C03631=1012.728,1.507,383.376,-29.710,62.357,-30.586
C03632=1012.729,1.110,383.407,-29.703,62.283,-30.592
C03633=1012.732,0.714,383.438,-29.696,62.210,-30.597
C03634=1012.733,0.320,383.469,-29.689,62.138,-30.603
C03635=1012.735,-0.076,383.499,-29.682,62.066,-30.609
C03636=1012.736,-0.474,383.530,-29.675,61.994,-30.616
C03637=1012.738,-0.874,383.560,-29.669,61.922,-30.622
C03638=1012.740,-1.277,383.591,-29.662,61.851,-30.627
C03639=1012.742,-1.681,383.623,-29.655,61.779,-30.634
C03640=1012.744,-2.088,383.654,-29.648,61.709,-30.640
C03641=1012.745,-2.496,383.686,-29.642,61.639,-30.646
C03642=1012.746,-2.906,383.717,-29.635,61.568,-30.653
C03643=1012.748,-3.317,383.749,-29.629,61.499,-30.660
C03644=1012.750,-3.719,383.781,-29.623,61.431,-30.667
C03645=1012.751,-4.104,383.810,-29.618,61.367,-30.674
C03646=1012.753,-4.484,383.839,-29.612,61.304,-30.679
C03647=1012.754,-4.874,383.869,-29.606,61.241,-30.686
C03648=1012.756,-5.289,383.902,-29.600,61.175,-30.693
C03649=1012.757,-5.503,383.919,-29.597,61.140,-30.697
C03650=1012.757,-5.720,383.935,-29.594,61.106,-30.699
C03651=1012.758,-5.936,383.952,-29.591,61.072,-30.704
C03652=1012.760,-6.154,383.969,-29.588,61.037,-30.708
C03653=1012.760,-6.370,383.986,-29.585,61.003,-30.710
C03654=1012.761,-6.586,384.002,-29.582,60.969,-30.715
C03655=1012.761,-6.803,384.019,-29.579,60.936,-30.719
C03656=1012.763,-7.019,384.036,-29.576,60.903,-30.722
C03657=1012.763,-7.233,384.052,-29.573,60.870,-30.726
C03658=1012.764,-7.448,384.069,-29.571,60.838,-30.730
C03659=1012.765,-7.661,384.085,-29.568,60.805,-30.734
C03660=1012.766,-7.874,384.102,-29.565,60.773,-30.736
C03661=1012.766,-8.086,384.118,-29.563,60.742,-30.742
C03662=1012.767,-8.297,384.135,-29.560,60.710,-30.745
C03663=1012.768,-8.509,384.150,-29.557,60.679,-30.748
C03664=1012.769,-8.721,384.167,-29.555,60.648,-30.752
C03665=1012.769,-8.932,384.183,-29.552,60.618,-30.756
C03666=1012.770,-9.143,384.200,-29.550,60.587,-30.759
C03667=1012.772,-9.564,384.233,-29.545,60.526,-30.767
C03668=1012.773,-9.986,384.265,-29.540,60.466,-30.775
C03669=1012.775,-10.407,384.298,-29.534,60.407,-30.781
C03670=1012.776,-10.827,384.331,-29.530,60.348,-30.789
C03671=1012.778,-11.244,384.363,-29.525,60.292,-30.796
C03672=1012.779,-11.662,384.395,-29.521,60.235,-30.804
C03673=1012.780,-12.078,384.427,-29.516,60.179,-30.811
C03674=1012.782,-12.491,384.459,-29.512,60.125,-30.818
C03675=1012.783,-12.903,384.491,-29.507,60.071,-30.825
C03676=1012.784,-13.307,384.523,-29.503,60.020,-30.833
C03677=1012.786,-13.699,384.553,-29.499,59.970,-30.839
C03678=1012.787,-14.081,384.582,-29.495,59.922,-30.846
C03679=1012.788,-14.456,384.611,-29.492,59.877,-30.853
C03680=1012.789,-14.832,384.640,-29.488,59.831,-30.859
C03681=1012.790,-15.211,384.670,-29.485,59.785,-30.866
C03682=1012.791,-15.599,384.700,-29.481,59.740,-30.873
C03683=1012.792,-15.994,384.730,-29.478,59.694,-30.880
C03684=1012.793,-16.390,384.761,-29.474,59.648,-30.887
C03685=1012.795,-16.786,384.791,-29.471,59.603,-30.894
C03686=1012.796,-17.184,384.822,-29.468,59.560,-30.901
C03687=1012.797,-17.573,384.852,-29.464,59.517,-30.907
C03688=1012.797,-17.970,384.884,-29.461,59.474,-30.914
C03689=1012.798,-18.197,384.901,-29.459,59.449,-30.917
C03690=1012.799,-18.450,384.920,-29.457,59.423,-30.922
C03691=1012.800,-18.721,384.942,-29.455,59.394,-30.926
C03692=1012.800,-19.000,384.964,-29.453,59.366,-30.931
C03693=1012.801,-19.275,384.984,-29.451,59.338,-30.936
C03694=1012.802,-19.532,385.004,-29.449,59.312,-30.941
C03695=1012.803,-19.762,385.022,-29.448,59.289,-30.944
C03696=1012.802,-19.967,385.038,-29.446,59.269,-30.948
C03697=1012.804,-20.318,385.065,-29.444,59.235,-30.954
C03698=1012.804,-20.714,385.096,-29.441,59.196,-30.961
C03699=1012.806,-21.107,385.127,-29.439,59.160,-30.967
C03700=1012.806,-21.501,385.157,-29.436,59.123,-30.974
C03701=1012.808,-21.894,385.187,-29.433,59.087,-30.980
C03702=1012.809,-22.287,385.218,-29.431,59.052,-30.987
C03703=1012.809,-22.680,385.248,-29.429,59.018,-30.992
C03704=1012.810,-23.074,385.279,-29.426,58.985,-30.999
C03705=1012.811,-23.467,385.308,-29.424,58.951,-31.005
C03706=1012.811,-23.860,385.339,-29.422,58.919,-31.013
C03707=1012.812,-24.253,385.370,-29.420,58.887,-31.019
C03708=1012.813,-24.646,385.401,-29.418,58.858,-31.024
C03709=1012.815,-25.040,385.430,-29.416,58.827,-31.031
C03710=1012.815,-25.433,385.461,-29.415,58.798,-31.037
C03711=1012.816,-25.827,385.492,-29.413,58.768,-31.043
C03712=1012.816,-26.219,385.522,-29.411,58.741,-31.049
C03713=1012.817,-26.613,385.552,-29.410,58.714,-31.055
C03714=1012.818,-27.007,385.583,-29.408,58.687,-31.062
C03715=1012.819,-27.399,385.613,-29.407,58.661,-31.067
C03716=1012.819,-27.793,385.644,-29.405,58.636,-31.073
C03717=1012.820,-28.186,385.674,-29.404,58.611,-31.079
C03718=1012.820,-28.580,385.705,-29.403,58.588,-31.084
C03719=1012.821,-28.973,385.735,-29.401,58.565,-31.090
C03720=1012.822,-29.366,385.766,-29.400,58.541,-31.096
C03721=1012.823,-29.760,385.796,-29.399,58.520,-31.101
C03722=1012.823,-30.153,385.826,-29.398,58.499,-31.106
C03723=1012.823,-30.547,385.857,-29.397,58.479,-31.113
C03724=1012.824,-30.940,385.888,-29.396,58.459,-31.118
C03725=1012.825,-31.333,385.918,-29.396,58.440,-31.124
C03726=1012.825,-31.727,385.948,-29.394,58.422,-31.128
C03727=1012.826,-32.120,385.979,-29.394,58.404,-31.135
C03728=1012.826,-32.514,386.010,-29.393,58.388,-31.138
C03729=1012.826,-32.907,386.040,-29.393,58.372,-31.144
C03730=1012.827,-33.301,386.070,-29.393,58.357,-31.149
C03731=1012.828,-33.694,386.101,-29.392,58.342,-31.155
C03732=1012.827,-34.087,386.131,-29.392,58.329,-31.159
C03733=1012.828,-34.481,386.162,-29.391,58.315,-31.164
C03734=1012.828,-34.874,386.192,-29.391,58.303,-31.169
C03735=1012.829,-35.268,386.222,-29.391,58.291,-31.173
C03736=1012.829,-35.662,386.253,-29.391,58.280,-31.178
C03737=1012.829,-36.055,386.283,-29.391,58.269,-31.182
C03738=1012.830,-36.448,386.314,-29.391,58.260,-31.187
C03739=1012.830,-36.841,386.344,-29.391,58.251,-31.192
C03740=1012.830,-37.235,386.375,-29.392,58.243,-31.197
C03741=1012.830,-37.628,386.405,-29.392,58.236,-31.200
C03742=1012.831,-38.022,386.436,-29.392,58.229,-31.205
C03743=1012.831,-38.415,386.466,-29.393,58.223,-31.208
C03744=1012.831,-38.809,386.497,-29.393,58.218,-31.212
C03745=1012.831,-39.202,386.527,-29.394,58.214,-31.217
C03746=1012.832,-39.595,386.558,-29.395,58.209,-31.222
C03747=1012.831,-39.988,386.588,-29.396,58.207,-31.226
C03748=1012.831,-40.381,386.618,-29.396,58.205,-31.229
C03749=1012.832,-40.775,386.649,-29.397,58.202,-31.233
C03750=1012.832,-41.167,386.679,-29.398,58.201,-31.237
C03751=1012.832,-41.560,386.709,-29.399,58.202,-31.240
C03752=1012.832,-41.954,386.739,-29.400,58.203,-31.243
C03753=1012.833,-42.347,386.770,-29.401,58.204,-31.247
C03754=1012.832,-42.740,386.801,-29.402,58.206,-31.251
C03755=1012.832,-43.133,386.831,-29.404,58.209,-31.254
C03756=1012.832,-43.526,386.862,-29.405,58.212,-31.258
C03757=1012.832,-43.919,386.892,-29.407,58.217,-31.261
C03758=1012.832,-44.312,386.923,-29.408,58.222,-31.264
C03759=1012.832,-44.705,386.953,-29.410,58.228,-31.267
C03760=1012.832,-45.097,386.984,-29.411,58.234,-31.270
C03761=1012.832,-45.490,387.014,-29.413,58.242,-31.273
C03762=1012.832,-45.884,387.044,-29.414,58.250,-31.275
C03763=1012.832,-46.277,387.074,-29.417,58.258,-31.279
C03764=1012.831,-46.669,387.105,-29.419,58.269,-31.281
C03765=1012.832,-47.062,387.135,-29.421,58.279,-31.284
C03766=1012.832,-47.455,387.165,-29.423,58.289,-31.286
C03767=1012.831,-47.847,387.196,-29.425,58.302,-31.288
C03768=1012.831,-48.240,387.227,-29.427,58.314,-31.292
C03769=1012.831,-48.632,387.257,-29.430,58.327,-31.294
C03770=1012.830,-49.025,387.287,-29.432,58.342,-31.296
C03771=1012.830,-49.418,387.318,-29.434,58.357,-31.298
C03772=1012.830,-49.811,387.348,-29.437,58.372,-31.299
C03773=1012.830,-50.202,387.379,-29.440,58.388,-31.303
C03774=1012.829,-50.596,387.409,-29.442,58.404,-31.304
C03775=1012.828,-50.988,387.439,-29.445,58.423,-31.306
C03776=1012.828,-51.381,387.470,-29.448,58.442,-31.309
C03777=1012.828,-51.773,387.500,-29.451,58.460,-31.310
C03778=1012.828,-52.166,387.530,-29.454,58.481,-31.312
C03779=1012.827,-52.558,387.561,-29.457,58.502,-31.313
C03780=1012.827,-52.951,387.591,-29.460,58.523,-31.315
C03781=1012.826,-53.344,387.622,-29.464,58.545,-31.317
C03782=1012.826,-53.736,387.651,-29.467,58.569,-31.319
C03783=1012.825,-54.128,387.682,-29.470,58.592,-31.319
C03784=1012.825,-54.521,387.713,-29.474,58.616,-31.321
C03785=1012.825,-54.913,387.742,-29.477,58.642,-31.323
C03786=1012.824,-55.305,387.773,-29.481,58.668,-31.323
C03787=1012.823,-55.698,387.804,-29.485,58.696,-31.324
C03788=1012.823,-56.091,387.834,-29.488,58.723,-31.326
C03789=1012.822,-56.483,387.865,-29.492,58.752,-31.326
C03790=1012.822,-56.876,387.895,-29.496,58.781,-31.327
C03791=1012.821,-57.270,387.925,-29.500,58.810,-31.329
C03792=1012.820,-57.664,387.956,-29.504,58.841,-31.329
C03793=1012.820,-58.059,387.986,-29.509,58.872,-31.330
C03794=1012.820,-58.452,388.017,-29.513,58.905,-31.330
C03795=1012.818,-58.848,388.047,-29.517,58.938,-31.331
C03796=1012.818,-59.244,388.078,-29.522,58.972,-31.332
C03797=1012.818,-59.640,388.109,-29.526,59.007,-31.332
C03798=1012.817,-60.037,388.139,-29.531,59.042,-31.333
C03799=1012.816,-60.434,388.170,-29.536,59.079,-31.334
C03800=1012.815,-60.832,388.201,-29.541,59.117,-31.334
C03801=1012.814,-61.230,388.232,-29.546,59.155,-31.334
C03802=1012.814,-61.630,388.263,-29.551,59.194,-31.334
C03803=1012.813,-62.029,388.294,-29.556,59.234,-31.335
C03804=1012.812,-62.428,388.325,-29.561,59.274,-31.335
C03805=1012.811,-62.829,388.356,-29.567,59.316,-31.336
C03806=1012.810,-63.229,388.386,-29.572,59.358,-31.335
C03807=1012.809,-63.631,388.418,-29.578,59.402,-31.336
C03808=1012.808,-64.032,388.448,-29.584,59.446,-31.336
C03809=1012.808,-64.434,388.479,-29.589,59.490,-31.336
C03810=1012.806,-64.836,388.511,-29.595,59.537,-31.335
C03811=1012.806,-65.239,388.542,-29.601,59.583,-31.336
C03812=1012.805,-65.642,388.573,-29.607,59.631,-31.334
C03813=1012.804,-66.045,388.604,-29.613,59.679,-31.335
C03814=1012.803,-66.449,388.635,-29.620,59.728,-31.336
C03815=1012.802,-66.852,388.667,-29.626,59.778,-31.334
C03816=1012.801,-67.256,388.698,-29.633,59.830,-31.334
C03817=1012.800,-67.661,388.730,-29.639,59.881,-31.334
C03818=1012.799,-68.065,388.761,-29.646,59.933,-31.334
C03819=1012.797,-68.468,388.792,-29.653,59.986,-31.333
C03820=1012.797,-68.872,388.824,-29.659,60.041,-31.332
C03821=1012.795,-69.277,388.855,-29.667,60.096,-31.332
C03822=1012.794,-69.681,388.886,-29.674,60.151,-31.332
C03823=1012.793,-70.085,388.917,-29.681,60.208,-31.332
C03824=1012.792,-70.490,388.949,-29.688,60.265,-31.331
C03825=1012.791,-70.894,388.980,-29.696,60.324,-31.330
C03826=1012.789,-71.298,389.011,-29.704,60.383,-31.330
C03827=1012.789,-71.702,389.042,-29.711,60.442,-31.330
C03828=1012.787,-72.106,389.074,-29.719,60.502,-31.329
C03829=1012.786,-72.510,389.105,-29.727,60.564,-31.330
C03830=1012.785,-72.914,389.136,-29.735,60.626,-31.328
C03831=1012.783,-73.317,389.168,-29.743,60.689,-31.328
C03832=1012.783,-73.721,389.199,-29.752,60.753,-31.329
C03833=1012.782,-74.124,389.230,-29.760,60.817,-31.328
C03834=1012.780,-74.527,389.262,-29.768,60.883,-31.326
C03835=1012.778,-74.930,389.293,-29.777,60.949,-31.327
C03836=1012.777,-75.333,389.324,-29.786,61.016,-31.327
C03837=1012.776,-75.737,389.355,-29.794,61.083,-31.325
C03838=1012.774,-76.139,389.387,-29.803,61.152,-31.325
C03839=1012.773,-76.541,389.417,-29.812,61.221,-31.324
C03840=1012.772,-76.944,389.449,-29.822,61.292,-31.324
C03841=1012.770,-77.345,389.480,-29.831,61.361,-31.323
C03842=1012.770,-77.747,389.511,-29.840,61.433,-31.324
C03843=1012.768,-78.149,389.542,-29.850,61.505,-31.324
C03844=1012.766,-78.550,389.573,-29.859,61.579,-31.322
C03845=1012.765,-78.950,389.604,-29.869,61.652,-31.323
C03846=1012.763,-79.351,389.636,-29.879,61.726,-31.322
C03847=1012.762,-79.751,389.666,-29.889,61.801,-31.323
C03848=1012.761,-80.150,389.697,-29.899,61.877,-31.323
C03849=1012.759,-80.549,389.728,-29.910,61.954,-31.323
C03850=1012.758,-80.946,389.759,-29.920,62.031,-31.322
C03851=1012.757,-81.344,389.790,-29.931,62.108,-31.323
C03852=1012.755,-81.741,389.820,-29.941,62.187,-31.323
C03853=1012.753,-82.140,389.851,-29.952,62.266,-31.322
C03854=1012.751,-82.538,389.882,-29.963,62.347,-31.323
C03855=1012.751,-82.934,389.913,-29.974,62.427,-31.324
C03856=1012.749,-83.330,389.944,-29.985,62.509,-31.323
C03857=1012.747,-83.726,389.975,-29.997,62.591,-31.324
C03858=1012.745,-84.117,390.005,-30.008,62.673,-31.325
C03859=1012.744,-84.509,390.035,-30.020,62.755,-31.325
C03860=1012.743,-84.928,390.068,-30.032,62.845,-31.325
C03861=1012.742,-85.158,390.086,-30.039,62.894,-31.326
C03862=1012.741,-85.395,390.104,-30.046,62.945,-31.326
C03863=1012.740,-85.635,390.122,-30.054,62.996,-31.328
C03864=1012.739,-85.869,390.141,-30.061,63.047,-31.328
C03865=1012.738,-86.093,390.158,-30.068,63.097,-31.329
C03866=1012.737,-86.500,390.190,-30.081,63.187,-31.330
C03867=1012.735,-86.887,390.220,-30.094,63.273,-31.332
C03868=1012.733,-87.264,390.249,-30.105,63.357,-31.332
C03869=1012.731,-87.633,390.277,-30.117,63.441,-31.333
C03870=1012.730,-87.995,390.306,-30.130,63.523,-31.335
C03871=1012.729,-88.372,390.336,-30.142,63.610,-31.336
C03872=1012.727,-88.756,390.364,-30.156,63.699,-31.339
C03873=1012.726,-88.975,390.382,-30.163,63.750,-31.339
C03874=1012.725,-89.218,390.401,-30.172,63.807,-31.342
C03875=1012.724,-89.473,390.421,-30.181,63.867,-31.343
C03876=1012.723,-89.732,390.441,-30.190,63.928,-31.344
C03877=1012.722,-89.983,390.460,-30.198,63.988,-31.344
C03878=1012.720,-90.216,390.478,-30.207,64.044,-31.346
C03879=1012.720,-90.427,390.495,-30.214,64.094,-31.348
C03880=1012.719,-90.696,390.516,-30.224,64.159,-31.349
C03881=1012.718,-91.050,390.543,-30.238,64.245,-31.353
C03882=1012.716,-91.439,390.573,-30.252,64.340,-31.355
C03883=1012.714,-91.828,390.604,-30.267,64.436,-31.359
C03884=1012.712,-92.216,390.634,-30.282,64.532,-31.361
C03885=1012.711,-92.604,390.664,-30.297,64.629,-31.364
C03886=1012.708,-92.989,390.694,-30.312,64.726,-31.367
C03887=1012.708,-93.376,390.723,-30.328,64.824,-31.371
C03888=1012.706,-93.760,390.754,-30.343,64.922,-31.375
C03889=1012.704,-94.145,390.784,-30.359,65.021,-31.378
C03890=1012.702,-94.527,390.813,-30.375,65.120,-31.382
C03891=1012.700,-94.909,390.843,-30.391,65.220,-31.386
C03892=1012.699,-95.289,390.873,-30.407,65.319,-31.391
C03893=1012.697,-95.669,390.902,-30.424,65.419,-31.396
C03894=1012.695,-96.046,390.932,-30.440,65.520,-31.400
C03895=1012.694,-96.424,390.960,-30.458,65.621,-31.406
C03896=1012.692,-96.801,390.989,-30.474,65.723,-31.411
C03897=1012.690,-97.176,391.019,-30.492,65.824,-31.418
C03898=1012.689,-97.552,391.049,-30.509,65.928,-31.423
C03899=1012.688,-97.928,391.077,-30.527,66.031,-31.429
C03900=1012.685,-98.303,391.106,-30.545,66.134,-31.435
C03901=1012.684,-98.678,391.136,-30.564,66.239,-31.442
C03902=1012.682,-99.055,391.165,-30.582,66.345,-31.448
C03903=1012.680,-99.432,391.194,-30.601,66.451,-31.455
C03904=1012.679,-99.809,391.224,-30.621,66.557,-31.464
C03905=1012.677,-100.187,391.253,-30.641,66.666,-31.472
C03906=1012.675,-100.567,391.283,-30.660,66.775,-31.479
C03907=1012.673,-100.947,391.313,-30.681,66.885,-31.488
C03908=1012.672,-101.330,391.343,-30.701,66.996,-31.495
C03909=1012.670,-101.712,391.372,-30.722,67.108,-31.505
C03910=1012.668,-102.096,391.402,-30.744,67.220,-31.516
C03911=1012.666,-102.480,391.433,-30.765,67.334,-31.523
C03912=1012.665,-102.865,391.462,-30.788,67.449,-31.535
C03913=1012.663,-103.251,391.492,-30.811,67.564,-31.546
C03914=1012.661,-103.637,391.523,-30.833,67.680,-31.556
C03915=1012.659,-104.024,391.552,-30.856,67.797,-31.567
C03916=1012.657,-104.412,391.582,-30.880,67.915,-31.580
C03917=1012.655,-104.799,391.612,-30.904,68.034,-31.591
C03918=1012.654,-105.188,391.643,-30.929,68.154,-31.603
C03919=1012.652,-105.576,391.673,-30.955,68.274,-31.618
C03920=1012.651,-105.965,391.703,-30.980,68.395,-31.630
C03921=1012.649,-106.356,391.734,-31.006,68.517,-31.646
C03922=1012.647,-106.763,391.766,-31.034,68.645,-31.661
C03923=1012.645,-106.977,391.782,-31.049,68.713,-31.670
C03924=1012.644,-107.197,391.799,-31.064,68.784,-31.678
C03925=1012.644,-107.424,391.817,-31.080,68.856,-31.686
C03926=1012.643,-107.654,391.835,-31.096,68.929,-31.695
C03927=1012.642,-107.887,391.853,-31.113,69.003,-31.705
C03928=1012.641,-108.118,391.871,-31.129,69.078,-31.714
C03929=1012.639,-108.348,391.889,-31.146,69.152,-31.723
C03930=1012.638,-108.573,391.907,-31.163,69.224,-31.735
C03931=1012.637,-108.792,391.923,-31.179,69.296,-31.743
C03932=1012.635,-109.209,391.956,-31.211,69.431,-31.764
C03933=1012.633,-109.603,391.987,-31.241,69.560,-31.782
C03934=1012.632,-109.992,392.017,-31.272,69.688,-31.802
C03935=1012.630,-110.380,392.047,-31.303,69.816,-31.820
C03936=1012.629,-110.769,392.078,-31.334,69.946,-31.840
C03937=1012.627,-111.158,392.108,-31.367,70.075,-31.862
C03938=1012.625,-111.547,392.139,-31.400,70.206,-31.884
C03939=1012.623,-111.935,392.168,-31.434,70.337,-31.906
C03940=1012.621,-112.323,392.199,-31.468,70.469,-31.928
C03941=1012.620,-112.712,392.229,-31.503,70.601,-31.953
C03942=1012.617,-113.101,392.259,-31.538,70.735,-31.976
C03943=1012.616,-113.489,392.290,-31.575,70.868,-32.003
C03944=1012.614,-113.878,392.320,-31.612,71.002,-32.028
C03945=1012.612,-114.266,392.350,-31.649,71.137,-32.054
C03946=1012.611,-114.655,392.381,-31.688,71.273,-32.082
C03947=1012.609,-115.043,392.411,-31.727,71.409,-32.111
C03948=1012.608,-115.431,392.441,-31.767,71.547,-32.140
C03949=1012.606,-115.820,392.471,-31.808,71.684,-32.170
C03950=1012.603,-116.209,392.502,-31.849,71.822,-32.201
C03951=1012.603,-116.597,392.532,-31.892,71.961,-32.233
C03952=1012.600,-116.985,392.562,-31.936,72.100,-32.267
C03953=1012.599,-117.373,392.593,-31.981,72.240,-32.302
C03954=1012.597,-117.762,392.623,-32.026,72.380,-32.337
C03955=1012.595,-118.150,392.653,-32.072,72.522,-32.372
C03956=1012.594,-118.539,392.684,-32.120,72.663,-32.411
C03957=1012.592,-118.926,392.714,-32.168,72.805,-32.448
C03958=1012.591,-119.315,392.744,-32.218,72.947,-32.489
C03959=1012.589,-119.703,392.775,-32.268,73.091,-32.528
C03960=1012.587,-120.091,392.804,-32.320,73.235,-32.571
C03961=1012.586,-120.480,392.835,-32.372,73.379,-32.613
C03962=1012.584,-120.867,392.866,-32.427,73.524,-32.660
C03963=1012.582,-121.256,392.895,-32.482,73.670,-32.704
C03964=1012.581,-121.644,392.926,-32.539,73.815,-32.752
C03965=1012.579,-122.032,392.956,-32.597,73.962,-32.801
C03966=1012.578,-122.420,392.987,-32.656,74.109,-32.852
C03967=1012.576,-122.808,393.017,-32.717,74.257,-32.903
C03968=1012.574,-123.197,393.047,-32.780,74.405,-32.957
C03969=1012.573,-123.584,393.077,-32.843,74.553,-33.012
C03970=1012.571,-123.972,393.108,-32.909,74.703,-33.069
C03971=1012.571,-124.360,393.138,-32.976,74.852,-33.127
C03972=1012.568,-124.749,393.168,-33.044,75.002,-33.187
C03973=1012.566,-125.136,393.199,-33.115,75.152,-33.249
C03974=1012.566,-125.525,393.229,-33.188,75.304,-33.315
C03975=1012.564,-125.912,393.259,-33.261,75.456,-33.379
C03976=1012.563,-126.300,393.290,-33.337,75.608,-33.447
C03977=1012.561,-126.688,393.319,-33.416,75.761,-33.519
C03978=1012.560,-127.076,393.350,-33.496,75.914,-33.591
C03979=1012.558,-127.464,393.380,-33.578,76.068,-33.666
C03980=1012.556,-127.853,393.410,-33.664,76.222,-33.745
C03981=1012.555,-128.240,393.441,-33.751,76.377,-33.824
C03982=1012.553,-128.628,393.471,-33.839,76.532,-33.905
C03983=1012.553,-129.016,393.501,-33.932,76.688,-33.991
C03984=1012.551,-129.404,393.531,-34.027,76.844,-34.079
C03985=1012.550,-129.792,393.562,-34.125,77.000,-34.171
C03986=1012.548,-130.180,393.592,-34.226,77.158,-34.265
C03987=1012.547,-130.568,393.623,-34.329,77.315,-34.362
C03988=1012.546,-130.955,393.652,-34.436,77.474,-34.462
C03989=1012.545,-131.343,393.683,-34.545,77.633,-34.565
C03990=1012.543,-131.731,393.713,-34.658,77.791,-34.672
C03991=1012.542,-132.119,393.744,-34.776,77.950,-34.785
C03992=1012.541,-132.507,393.773,-34.897,78.110,-34.899
C03993=1012.540,-132.895,393.804,-35.020,78.271,-35.016
C03994=1012.538,-133.282,393.834,-35.149,78.432,-35.139
C03995=1012.537,-133.671,393.864,-35.283,78.593,-35.269
C03996=1012.536,-134.058,393.894,-35.420,78.754,-35.401
C03997=1012.641,-134.083,393.455,-31.214,69.087,-31.893
C03998=1012.644,-133.696,393.425,-31.175,68.914,-31.872
C03999=1012.647,-133.308,393.395,-31.137,68.742,-31.852
C04000=1012.648,-132.920,393.364,-31.100,68.570,-31.833
C04001=1012.652,-132.532,393.334,-31.064,68.399,-31.816
C04002=1012.653,-132.145,393.304,-31.029,68.229,-31.799
C04003=1012.657,-131.757,393.274,-30.994,68.059,-31.783
C04004=1012.658,-131.369,393.244,-30.960,67.890,-31.767
C04005=1012.661,-130.981,393.213,-30.926,67.721,-31.752
C04006=1012.664,-130.593,393.183,-30.893,67.553,-31.739
C04007=1012.666,-130.206,393.153,-30.861,67.384,-31.726
C04008=1012.669,-129.818,393.123,-30.829,67.218,-31.714
C04009=1012.671,-129.429,393.093,-30.798,67.051,-31.703
C04010=1012.673,-129.042,393.062,-30.767,66.885,-31.691
C04011=1012.676,-128.654,393.032,-30.737,66.719,-31.681
C04012=1012.679,-128.266,393.002,-30.708,66.555,-31.672
C04013=1012.681,-127.879,392.972,-30.678,66.390,-31.662
C04014=1012.684,-127.490,392.942,-30.650,66.227,-31.655
C04015=1012.687,-127.102,392.912,-30.621,66.063,-31.647
C04016=1012.689,-126.715,392.881,-30.593,65.901,-31.639
C04017=1012.692,-126.327,392.851,-30.567,65.739,-31.633
C04018=1012.694,-125.939,392.821,-30.540,65.577,-31.628
C04019=1012.697,-125.551,392.791,-30.513,65.416,-31.622
C04020=1012.700,-125.162,392.760,-30.487,65.256,-31.617
C04021=1012.702,-124.775,392.731,-30.461,65.097,-31.612
C04022=1012.705,-124.387,392.700,-30.437,64.937,-31.610
C04023=1012.708,-123.999,392.670,-30.412,64.780,-31.605
C04024=1012.710,-123.611,392.639,-30.388,64.622,-31.603
C04025=1012.713,-123.222,392.609,-30.364,64.464,-31.601
C04026=1012.716,-122.835,392.579,-30.340,64.307,-31.599
C04027=1012.718,-122.447,392.549,-30.316,64.152,-31.597
C04028=1012.721,-122.059,392.519,-30.293,63.997,-31.596
C04029=1012.723,-121.670,392.489,-30.270,63.841,-31.595
C04030=1012.726,-121.282,392.459,-30.249,63.687,-31.597
C04031=1012.728,-120.894,392.428,-30.226,63.533,-31.596
C04032=1012.732,-120.506,392.398,-30.205,63.381,-31.597
C04033=1012.734,-120.118,392.368,-30.183,63.227,-31.598
C04034=1012.737,-119.730,392.338,-30.162,63.076,-31.599
C04035=1012.740,-119.342,392.307,-30.141,62.925,-31.601
C04036=1012.743,-118.954,392.277,-30.121,62.774,-31.604
C04037=1012.745,-118.565,392.247,-30.100,62.624,-31.606
C04038=1012.748,-118.177,392.217,-30.080,62.475,-31.608
C04039=1012.750,-117.789,392.187,-30.060,62.326,-31.612
C04040=1012.754,-117.401,392.157,-30.040,62.178,-31.614
C04041=1012.756,-117.012,392.127,-30.021,62.031,-31.620
C04042=1012.759,-116.624,392.097,-30.002,61.884,-31.623
C04043=1012.761,-116.236,392.066,-29.983,61.738,-31.628
C04044=1012.764,-115.848,392.036,-29.964,61.592,-31.633
C04045=1012.766,-115.459,392.006,-29.946,61.447,-31.638
C04046=1012.770,-115.070,391.976,-29.928,61.303,-31.644
C04047=1012.773,-114.682,391.945,-29.910,61.159,-31.648
C04048=1012.775,-114.293,391.915,-29.892,61.017,-31.655
C04049=1012.778,-113.905,391.885,-29.874,60.874,-31.661
C04050=1012.780,-113.517,391.855,-29.857,60.733,-31.666
C04051=1012.783,-113.128,391.826,-29.840,60.591,-31.674
C04052=1012.786,-112.739,391.795,-29.823,60.451,-31.681
C04053=1012.789,-112.351,391.765,-29.806,60.310,-31.688
C04054=1012.791,-111.962,391.735,-29.789,60.172,-31.696
C04055=1012.794,-111.574,391.704,-29.773,60.034,-31.702
C04056=1012.797,-111.185,391.675,-29.756,59.895,-31.711
C04057=1012.800,-110.797,391.644,-29.740,59.758,-31.719
C04058=1012.802,-110.408,391.615,-29.724,59.622,-31.726
C04059=1012.805,-110.019,391.584,-29.708,59.486,-31.734
C04060=1012.808,-109.630,391.554,-29.692,59.351,-31.743
C04061=1012.811,-109.237,391.523,-29.677,59.215,-31.752
C04062=1012.814,-108.819,391.491,-29.660,59.072,-31.761
C04063=1012.815,-108.600,391.474,-29.652,58.997,-31.767
C04064=1012.816,-108.375,391.456,-29.643,58.920,-31.772
C04065=1012.818,-108.146,391.439,-29.634,58.843,-31.776
C04066=1012.820,-107.914,391.421,-29.625,58.764,-31.782
C04067=1012.822,-107.682,391.402,-29.617,58.686,-31.789
C04068=1012.823,-107.451,391.385,-29.608,58.608,-31.796
C04069=1012.824,-107.225,391.368,-29.599,58.532,-31.801
C04070=1012.827,-107.004,391.350,-29.591,58.458,-31.807
C04071=1012.828,-106.790,391.333,-29.583,58.387,-31.812
C04072=1012.831,-106.383,391.302,-29.568,58.252,-31.821
C04073=1012.833,-105.993,391.272,-29.554,58.123,-31.832
C04074=1012.836,-105.604,391.242,-29.540,57.995,-31.842
C04075=1012.839,-105.216,391.212,-29.525,57.869,-31.852
C04076=1012.841,-104.827,391.182,-29.511,57.743,-31.862
C04077=1012.844,-104.440,391.152,-29.498,57.618,-31.874
C04078=1012.847,-104.052,391.122,-29.484,57.493,-31.884
C04079=1012.849,-103.665,391.092,-29.471,57.371,-31.894
C04080=1012.852,-103.279,391.062,-29.458,57.248,-31.906
C04081=1012.854,-102.893,391.032,-29.444,57.127,-31.916
C04082=1012.857,-102.508,391.002,-29.431,57.007,-31.926
C04083=1012.860,-102.123,390.973,-29.419,56.888,-31.938
C04084=1012.862,-101.741,390.943,-29.406,56.769,-31.949
C04085=1012.864,-101.357,390.914,-29.393,56.651,-31.960
C04086=1012.867,-100.976,390.884,-29.381,56.535,-31.971
C04087=1012.869,-100.595,390.855,-29.369,56.420,-31.983
C04088=1012.873,-100.216,390.825,-29.357,56.305,-31.994
C04089=1012.875,-99.838,390.796,-29.345,56.192,-32.006
C04090=1012.877,-99.460,390.767,-29.333,56.080,-32.017
C04091=1012.880,-99.084,390.738,-29.321,55.968,-32.027
C04092=1012.882,-98.707,390.709,-29.309,55.857,-32.040
C04093=1012.884,-98.331,390.680,-29.298,55.748,-32.050
C04094=1012.887,-97.958,390.651,-29.286,55.640,-32.061
C04095=1012.889,-97.582,390.622,-29.275,55.532,-32.073
C04096=1012.892,-97.205,390.592,-29.264,55.424,-32.085
C04097=1012.894,-96.828,390.564,-29.252,55.316,-32.095
C04098=1012.897,-96.452,390.534,-29.241,55.210,-32.107
C04099=1012.899,-96.075,390.506,-29.230,55.105,-32.120
C04100=1012.902,-95.697,390.476,-29.219,54.999,-32.132
C04101=1012.904,-95.317,390.447,-29.208,54.894,-32.143
C04102=1012.906,-94.938,390.418,-29.197,54.790,-32.155
C04103=1012.909,-94.556,390.389,-29.187,54.686,-32.167
C04104=1012.911,-94.173,390.358,-29.176,54.583,-32.178
C04105=1012.914,-93.789,390.329,-29.165,54.479,-32.191
C04106=1012.916,-93.404,390.300,-29.155,54.376,-32.203
C04107=1012.918,-93.018,390.270,-29.144,54.274,-32.215
C04108=1012.920,-92.632,390.240,-29.133,54.173,-32.226
C04109=1012.922,-92.244,390.210,-29.123,54.071,-32.239
C04110=1012.925,-91.856,390.180,-29.113,53.970,-32.251
C04111=1012.928,-91.468,390.150,-29.102,53.871,-32.262
C04112=1012.930,-91.079,390.120,-29.092,53.771,-32.275
C04113=1012.933,-90.725,390.093,-29.083,53.682,-32.287
C04114=1012.934,-90.456,390.073,-29.076,53.614,-32.294
C04115=1012.935,-90.245,390.056,-29.071,53.561,-32.301
C04116=1012.937,-90.011,390.038,-29.065,53.504,-32.308
C04117=1012.938,-89.761,390.018,-29.058,53.441,-32.315
C04118=1012.939,-89.502,389.999,-29.052,53.378,-32.323
C04119=1012.941,-89.246,389.979,-29.045,53.315,-32.332
C04120=1012.942,-89.004,389.960,-29.039,53.255,-32.339
C04121=1012.944,-88.785,389.943,-29.034,53.201,-32.346
C04122=1012.946,-88.400,389.913,-29.024,53.109,-32.358
C04123=1012.948,-88.023,389.885,-29.015,53.018,-32.369
C04124=1012.950,-87.661,389.857,-29.006,52.933,-32.380
C04125=1012.953,-87.293,389.828,-28.997,52.847,-32.391
C04126=1012.954,-86.916,389.799,-28.988,52.758,-32.402
C04127=1012.956,-86.528,389.770,-28.979,52.668,-32.414
C04128=1012.959,-86.121,389.738,-28.969,52.574,-32.426
C04129=1012.960,-85.898,389.721,-28.964,52.523,-32.433
C04130=1012.961,-85.664,389.703,-28.958,52.471,-32.439
C04131=1012.963,-85.424,389.685,-28.953,52.416,-32.447
C04132=1012.964,-85.187,389.666,-28.947,52.363,-32.453
C04133=1012.965,-84.958,389.648,-28.942,52.312,-32.460
C04134=1012.968,-84.538,389.616,-28.932,52.219,-32.473
C04135=1012.970,-84.146,389.586,-28.924,52.133,-32.484
C04136=1012.972,-83.755,389.556,-28.915,52.048,-32.496
C04137=1012.974,-83.359,389.525,-28.906,51.963,-32.507
C04138=1012.976,-82.962,389.495,-28.897,51.878,-32.519
C04139=1012.978,-82.567,389.464,-28.889,51.795,-32.530
C04140=1012.979,-82.169,389.434,-28.880,51.711,-32.542
C04141=1012.982,-81.770,389.403,-28.872,51.629,-32.552
C04142=1012.984,-81.372,389.372,-28.863,51.547,-32.564
C04143=1012.986,-80.976,389.342,-28.855,51.467,-32.573
C04144=1012.987,-80.578,389.311,-28.847,51.386,-32.585
C04145=1012.991,-80.179,389.280,-28.838,51.307,-32.596
C04146=1012.992,-79.780,389.250,-28.830,51.229,-32.607
C04147=1012.993,-79.380,389.219,-28.822,51.151,-32.617
C04148=1012.996,-78.980,389.188,-28.814,51.074,-32.627
C04149=1012.998,-78.579,389.157,-28.806,50.998,-32.639
C04150=1012.999,-78.178,389.126,-28.798,50.922,-32.648
C04151=1013.001,-77.776,389.095,-28.790,50.847,-32.659
C04152=1013.003,-77.375,389.064,-28.783,50.772,-32.670
C04153=1013.005,-76.972,389.033,-28.775,50.699,-32.680
C04154=1013.006,-76.570,389.003,-28.768,50.627,-32.689
C04155=1013.009,-76.168,388.971,-28.760,50.556,-32.700
C04156=1013.011,-75.766,388.940,-28.753,50.485,-32.710
C04157=1013.012,-75.363,388.909,-28.745,50.414,-32.719
C04158=1013.014,-74.959,388.878,-28.738,50.345,-32.728
C04159=1013.016,-74.556,388.848,-28.731,50.277,-32.739
C04160=1013.017,-74.153,388.816,-28.724,50.209,-32.748
C04161=1013.020,-73.750,388.785,-28.717,50.142,-32.757
C04162=1013.021,-73.347,388.754,-28.710,50.076,-32.766
C04163=1013.023,-72.943,388.723,-28.703,50.011,-32.775
C04164=1013.025,-72.539,388.692,-28.696,49.948,-32.783
C04165=1013.026,-72.136,388.661,-28.690,49.884,-32.793
C04166=1013.027,-71.732,388.630,-28.683,49.822,-32.801
C04167=1013.029,-71.328,388.599,-28.676,49.760,-32.809
C04168=1013.030,-70.923,388.568,-28.670,49.699,-32.817
C04169=1013.032,-70.519,388.537,-28.664,49.638,-32.826
C04170=1013.033,-70.115,388.506,-28.657,49.579,-32.834
C04171=1013.035,-69.711,388.474,-28.651,49.521,-32.842
C04172=1013.036,-69.307,388.443,-28.645,49.463,-32.849
C04173=1013.038,-68.903,388.412,-28.639,49.407,-32.857
C04174=1013.039,-68.498,388.381,-28.633,49.351,-32.864
C04175=1013.041,-68.094,388.350,-28.627,49.296,-32.872
C04176=1013.042,-67.690,388.319,-28.621,49.242,-32.879
C04177=1013.044,-67.286,388.288,-28.615,49.189,-32.886
C04178=1013.045,-66.881,388.257,-28.610,49.136,-32.893
C04179=1013.047,-66.479,388.225,-28.604,49.084,-32.900
C04180=1013.048,-66.075,388.195,-28.599,49.034,-32.906
C04181=1013.049,-65.672,388.163,-28.593,48.984,-32.913
C04182=1013.050,-65.269,388.132,-28.588,48.935,-32.918
C04183=1013.052,-64.867,388.101,-28.583,48.887,-32.926
C04184=1013.053,-64.464,388.070,-28.578,48.841,-32.931
C04185=1013.054,-64.062,388.039,-28.573,48.794,-32.937
C04186=1013.055,-63.660,388.008,-28.568,48.748,-32.942
C04187=1013.056,-63.259,387.977,-28.563,48.704,-32.947
C04188=1013.057,-62.859,387.947,-28.558,48.661,-32.952
C04189=1013.058,-62.458,387.916,-28.553,48.618,-32.958
C04190=1013.059,-62.058,387.884,-28.549,48.576,-32.963
C04191=1013.061,-61.659,387.854,-28.544,48.534,-32.967
C04192=1013.062,-61.260,387.823,-28.540,48.495,-32.972
C04193=1013.063,-60.862,387.793,-28.535,48.456,-32.977
C04194=1013.064,-60.464,387.762,-28.531,48.416,-32.981
C04195=1013.065,-60.067,387.731,-28.527,48.379,-32.985
C04196=1013.066,-59.670,387.700,-28.523,48.343,-32.989
C04197=1013.067,-59.273,387.670,-28.519,48.307,-32.992
C04198=1013.067,-58.878,387.640,-28.515,48.272,-32.996
C04199=1013.068,-58.483,387.609,-28.511,48.238,-32.999
C04200=1013.069,-58.089,387.579,-28.507,48.204,-33.002
C04201=1013.070,-57.694,387.548,-28.503,48.172,-33.005
C04202=1013.071,-57.300,387.518,-28.500,48.141,-33.008
C04203=1013.072,-56.907,387.488,-28.496,48.110,-33.011
C04204=1013.072,-56.514,387.457,-28.493,48.079,-33.013
C04205=1013.074,-56.121,387.427,-28.489,48.050,-33.016
C04206=1013.074,-55.728,387.396,-28.486,48.023,-33.018
C04207=1013.075,-55.336,387.367,-28.483,47.995,-33.020
C04208=1013.075,-54.944,387.336,-28.480,47.967,-33.022
C04209=1013.076,-54.551,387.306,-28.477,47.941,-33.024
C04210=1013.076,-54.158,387.275,-28.474,47.916,-33.026
C04211=1013.078,-53.766,387.245,-28.471,47.892,-33.027
C04212=1013.078,-53.374,387.216,-28.468,47.869,-33.028
C04213=1013.078,-52.982,387.185,-28.465,47.846,-33.028
C04214=1013.078,-52.588,387.155,-28.462,47.824,-33.029
C04215=1013.080,-52.196,387.124,-28.460,47.803,-33.030
C04216=1013.080,-51.803,387.094,-28.457,47.782,-33.031
C04217=1013.080,-51.412,387.064,-28.455,47.762,-33.031
C04218=1013.081,-51.019,387.034,-28.452,47.743,-33.031
C04219=1013.081,-50.626,387.003,-28.450,47.726,-33.031
C04220=1013.082,-50.233,386.973,-28.448,47.708,-33.031
C04221=1013.082,-49.841,386.942,-28.446,47.691,-33.030
C04222=1013.082,-49.448,386.912,-28.444,47.675,-33.029
C04223=1013.083,-49.056,386.882,-28.442,47.660,-33.029
C04224=1013.083,-48.663,386.852,-28.440,47.646,-33.028
C04225=1013.084,-48.270,386.821,-28.438,47.633,-33.027
C04226=1013.083,-47.878,386.791,-28.436,47.620,-33.025
C04227=1013.085,-47.486,386.761,-28.434,47.608,-33.024
C04228=1013.085,-47.093,386.730,-28.433,47.597,-33.023
C04229=1013.085,-46.700,386.700,-28.431,47.587,-33.021
C04230=1013.085,-46.308,386.669,-28.430,47.577,-33.019
C04231=1013.085,-45.915,386.639,-28.428,47.568,-33.016
C04232=1013.085,-45.521,386.609,-28.427,47.559,-33.015
C04233=1013.086,-45.129,386.578,-28.426,47.552,-33.011
C04234=1013.086,-44.736,386.548,-28.425,47.547,-33.009
C04235=1013.086,-44.343,386.518,-28.424,47.541,-33.006
C04236=1013.085,-43.950,386.488,-28.422,47.535,-33.003
C04237=1013.086,-43.557,386.457,-28.422,47.531,-33.000
C04238=1013.086,-43.165,386.426,-28.421,47.527,-32.997
C04239=1013.086,-42.771,386.396,-28.420,47.525,-32.993
C04240=1013.086,-42.378,386.365,-28.419,47.523,-32.990
C04241=1013.086,-41.985,386.335,-28.419,47.521,-32.987
C04242=1013.086,-41.592,386.305,-28.418,47.521,-32.982
C04243=1013.085,-41.198,386.274,-28.418,47.521,-32.978
C04244=1013.086,-40.805,386.244,-28.417,47.522,-32.973
C04245=1013.085,-40.413,386.214,-28.417,47.525,-32.969
C04246=1013.085,-40.019,386.183,-28.416,47.526,-32.964
C04247=1013.085,-39.626,386.153,-28.416,47.531,-32.959
C04248=1013.085,-39.233,386.123,-28.416,47.535,-32.955
C04249=1013.084,-38.840,386.092,-28.416,47.540,-32.948
C04250=1013.084,-38.446,386.062,-28.416,47.546,-32.943
C04251=1013.084,-38.053,386.031,-28.416,47.551,-32.938
C04252=1013.084,-37.660,386.000,-28.416,47.558,-32.933
C04253=1013.083,-37.266,385.970,-28.417,47.566,-32.927
C04254=1013.083,-36.873,385.940,-28.417,47.576,-32.920
C04255=1013.083,-36.479,385.909,-28.417,47.585,-32.914
C04256=1013.082,-36.086,385.878,-28.417,47.595,-32.907
C04257=1013.082,-35.693,385.848,-28.418,47.606,-32.902
C04258=1013.082,-35.299,385.817,-28.419,47.618,-32.895
C04259=1013.082,-34.906,385.787,-28.419,47.629,-32.888
C04260=1013.081,-34.513,385.757,-28.420,47.643,-32.881
C04261=1013.080,-34.119,385.726,-28.421,47.657,-32.874
C04262=1013.079,-33.726,385.696,-28.422,47.672,-32.865
C04263=1013.079,-33.333,385.665,-28.423,47.687,-32.859
C04264=1013.079,-32.939,385.635,-28.424,47.703,-32.852
C04265=1013.078,-32.546,385.604,-28.424,47.720,-32.843
C04266=1013.077,-32.152,385.574,-28.426,47.737,-32.834
C04267=1013.078,-31.759,385.543,-28.427,47.756,-32.827
C04268=1013.076,-31.366,385.513,-28.428,47.775,-32.818
C04269=1013.076,-30.972,385.482,-28.429,47.795,-32.810
C04270=1013.075,-30.578,385.452,-28.431,47.815,-32.801
C04271=1013.074,-30.185,385.421,-28.432,47.837,-32.792
C04272=1013.073,-29.792,385.391,-28.434,47.859,-32.783
C04273=1013.073,-29.399,385.360,-28.435,47.881,-32.775
C04274=1013.073,-29.005,385.330,-28.437,47.905,-32.765
C04275=1013.072,-28.611,385.299,-28.439,47.929,-32.756
C04276=1013.071,-28.219,385.269,-28.440,47.954,-32.746
C04277=1013.070,-27.825,385.238,-28.442,47.980,-32.737
C04278=1013.070,-27.432,385.207,-28.444,48.006,-32.727
C04279=1013.068,-27.038,385.178,-28.446,48.033,-32.717
C04280=1013.067,-26.645,385.147,-28.448,48.061,-32.706
C04281=1013.066,-26.252,385.116,-28.450,48.090,-32.697
C04282=1013.066,-25.859,385.085,-28.453,48.119,-32.686
C04283=1013.065,-25.466,385.055,-28.455,48.149,-32.675
C04284=1013.064,-25.072,385.025,-28.457,48.179,-32.665
C04285=1013.062,-24.679,384.994,-28.459,48.211,-32.654
C04286=1013.062,-24.286,384.963,-28.462,48.243,-32.643
C04287=1013.061,-23.893,384.933,-28.464,48.275,-32.633
C04288=1013.060,-23.500,384.902,-28.467,48.309,-32.621
C04289=1013.058,-23.106,384.872,-28.470,48.343,-32.610
C04290=1013.057,-22.713,384.841,-28.472,48.378,-32.598
C04291=1013.056,-22.320,384.810,-28.475,48.414,-32.586
C04292=1013.055,-21.927,384.780,-28.478,48.450,-32.574
C04293=1013.054,-21.533,384.749,-28.480,48.488,-32.562
C04294=1013.053,-21.140,384.719,-28.483,48.526,-32.550
C04295=1013.052,-20.747,384.689,-28.486,48.564,-32.538
C04296=1013.050,-20.351,384.658,-28.489,48.604,-32.525
C04297=1013.049,-20.000,384.630,-28.492,48.639,-32.515
C04298=1013.049,-19.795,384.614,-28.494,48.661,-32.508
C04299=1013.048,-19.564,384.596,-28.495,48.684,-32.501
C04300=1013.047,-19.308,384.576,-28.498,48.712,-32.493
C04301=1013.046,-19.034,384.555,-28.500,48.741,-32.484
C04302=1013.046,-18.755,384.533,-28.502,48.770,-32.475
C04303=1013.044,-18.483,384.512,-28.504,48.800,-32.466
C04304=1013.043,-18.230,384.493,-28.507,48.827,-32.458
C04305=1013.043,-18.003,384.476,-28.509,48.853,-32.450
C04306=1013.041,-17.606,384.444,-28.512,48.897,-32.437
C04307=1013.040,-17.217,384.414,-28.515,48.941,-32.424
C04308=1013.038,-16.819,384.383,-28.519,48.988,-32.411
C04309=1013.038,-16.423,384.352,-28.523,49.035,-32.396
C04310=1013.036,-16.027,384.321,-28.526,49.082,-32.383
C04311=1013.034,-15.632,384.291,-28.530,49.130,-32.369
C04312=1013.033,-15.245,384.261,-28.534,49.176,-32.357
C04313=1013.032,-14.865,384.232,-28.537,49.224,-32.342
C04314=1013.030,-14.490,384.203,-28.541,49.272,-32.328
C04315=1013.029,-14.115,384.173,-28.544,49.320,-32.314
C04316=1013.028,-13.733,384.143,-28.548,49.369,-32.301
C04317=1013.025,-13.341,384.112,-28.552,49.421,-32.287
C04318=1013.024,-12.937,384.082,-28.557,49.475,-32.271
C04319=1013.022,-12.525,384.050,-28.561,49.530,-32.257
C04320=1013.021,-12.112,384.018,-28.565,49.586,-32.242
C04321=1013.019,-11.696,383.985,-28.570,49.644,-32.226
C04322=1013.018,-11.279,383.952,-28.574,49.702,-32.211
C04323=1013.015,-10.861,383.920,-28.579,49.762,-32.194
C04324=1013.014,-10.441,383.887,-28.584,49.823,-32.179
C04325=1013.012,-10.021,383.854,-28.588,49.884,-32.162
C04326=1013.010,-9.599,383.822,-28.593,49.946,-32.145
C04327=1013.008,-9.177,383.789,-28.598,50.009,-32.130
C04328=1013.007,-8.966,383.773,-28.601,50.041,-32.122
C04329=1013.006,-8.755,383.757,-28.603,50.073,-32.113
C04330=1013.005,-8.544,383.740,-28.605,50.105,-32.105
C04331=1013.004,-8.332,383.723,-28.608,50.138,-32.097
C04332=1013.003,-8.048,383.701,-28.611,50.181,-32.086
C04333=1013.001,-7.695,383.673,-28.616,50.237,-32.072
C04334=1012.999,-7.482,383.657,-28.618,50.270,-32.063
C04335=1012.999,-7.268,383.640,-28.621,50.304,-32.055
C04336=1012.998,-7.052,383.624,-28.623,50.339,-32.046
C04337=1012.997,-6.837,383.607,-28.626,50.373,-32.038
C04338=1012.996,-6.621,383.590,-28.629,50.407,-32.029
C04339=1012.995,-6.404,383.573,-28.631,50.442,-32.019
C04340=1012.994,-6.187,383.556,-28.634,50.478,-32.012
C04341=1012.993,-5.970,383.539,-28.637,50.514,-32.003
C04342=1012.992,-5.754,383.523,-28.639,50.549,-31.993
C04343=1012.991,-5.538,383.506,-28.642,50.584,-31.985
C04344=1012.989,-5.323,383.489,-28.645,50.620,-31.976
C04345=1012.989,-5.113,383.473,-28.648,50.655,-31.969
C04346=1012.987,-4.711,383.442,-28.653,50.723,-31.951
C04347=1012.985,-4.328,383.412,-28.658,50.788,-31.936
C04348=1012.982,-3.948,383.382,-28.663,50.854,-31.919
C04349=1012.981,-3.555,383.352,-28.668,50.921,-31.903
C04350=1012.979,-3.146,383.319,-28.674,50.994,-31.886
C04351=1012.977,-2.735,383.288,-28.679,51.066,-31.870
C04352=1012.974,-2.326,383.256,-28.685,51.140,-31.852
C04353=1012.972,-1.919,383.224,-28.690,51.213,-31.835
C04354=1012.970,-1.513,383.193,-28.696,51.286,-31.818
C04355=1012.968,-1.110,383.161,-28.702,51.361,-31.801
C04356=1012.966,-0.708,383.130,-28.707,51.434,-31.785
C04357=1012.964,-0.309,383.099,-28.713,51.509,-31.767
C04358=1012.961,0.087,383.069,-28.719,51.584,-31.750
C04359=1012.960,0.482,383.038,-28.724,51.659,-31.734
C04360=1012.957,0.876,383.007,-28.730,51.735,-31.717
C04361=1012.955,1.273,382.976,-28.736,51.812,-31.700
C04362=1012.952,1.669,382.945,-28.742,51.889,-31.682
C04363=1012.950,2.053,382.915,-28.747,51.964,-31.666
C04364=1012.949,2.409,382.888,-28.753,52.034,-31.651
C04365=1012.946,2.740,382.862,-28.758,52.100,-31.637
C04366=1012.944,3.060,382.837,-28.763,52.166,-31.623
C04367=1012.943,3.392,382.810,-28.768,52.232,-31.607
C04368=1012.941,3.751,382.783,-28.773,52.305,-31.593
C04369=1012.938,4.135,382.753,-28.779,52.385,-31.576
C04370=1012.936,4.526,382.723,-28.785,52.465,-31.558
C04371=1012.934,4.915,382.693,-28.792,52.546,-31.543
C04372=1012.931,5.304,382.662,-28.798,52.627,-31.526
C04373=1012.929,5.696,382.632,-28.804,52.711,-31.508
C04374=1012.926,6.089,382.601,-28.810,52.794,-31.491
C04375=1012.924,6.481,382.571,-28.816,52.878,-31.474
C04376=1012.921,6.869,382.540,-28.823,52.962,-31.457
C04377=1012.920,7.253,382.511,-28.829,53.045,-31.440
C04378=1012.916,7.633,382.481,-28.835,53.128,-31.425
C04379=1012.915,8.010,382.452,-28.842,53.211,-31.408
C04380=1012.912,8.384,382.423,-28.848,53.295,-31.391
C04381=1012.910,8.758,382.394,-28.854,53.379,-31.374
C04382=1012.907,9.131,382.365,-28.860,53.463,-31.358
C04383=1012.905,9.505,382.336,-28.867,53.547,-31.343
C04384=1012.903,9.881,382.306,-28.873,53.632,-31.327
C04385=1012.900,10.257,382.277,-28.879,53.719,-31.309
C04386=1012.897,10.635,382.248,-28.886,53.806,-31.294
C04387=1012.895,11.004,382.219,-28.893,53.892,-31.277
C04388=1012.893,11.367,382.191,-28.899,53.976,-31.262
C04389=1012.891,11.733,382.163,-28.905,54.062,-31.246
C04390=1012.888,12.111,382.133,-28.912,54.152,-31.229
C04391=1012.885,12.496,382.104,-28.919,54.243,-31.214
C04392=1012.883,12.880,382.073,-28.926,54.335,-31.197
C04393=1012.881,13.263,382.044,-28.933,54.428,-31.180
C04394=1012.877,13.644,382.014,-28.940,54.520,-31.164
C04395=1012.875,14.026,381.984,-28.947,54.613,-31.148
C04396=1012.873,14.406,381.955,-28.954,54.706,-31.133
C04397=1012.870,14.787,381.925,-28.961,54.800,-31.116
C04398=1012.867,15.166,381.896,-28.968,54.894,-31.100
C04399=1012.864,15.547,381.866,-28.975,54.989,-31.083
C04400=1012.862,15.928,381.837,-28.983,55.085,-31.067
C04401=1012.859,16.310,381.807,-28.990,55.181,-31.051
C04402=1012.857,16.693,381.778,-28.997,55.278,-31.035
C04403=1012.854,17.078,381.747,-29.005,55.377,-31.018
C04404=1012.851,17.465,381.717,-29.012,55.476,-31.003
C04405=1012.848,17.853,381.687,-29.020,55.576,-30.986
C04406=1012.846,18.245,381.657,-29.028,55.678,-30.971
C04407=1012.843,18.636,381.627,-29.036,55.780,-30.955
C04408=1012.840,19.041,381.595,-29.044,55.885,-30.938
C04409=1012.838,19.321,381.574,-29.049,55.960,-30.927
C04410=1012.835,19.668,381.546,-29.056,56.051,-30.913
C04411=1012.834,19.909,381.528,-29.061,56.116,-30.902
C04412=1012.832,20.170,381.507,-29.067,56.185,-30.892
C04413=1012.830,20.439,381.487,-29.072,56.257,-30.881
C04414=1012.828,20.707,381.466,-29.078,56.328,-30.871
C04415=1012.826,20.967,381.445,-29.083,56.399,-30.860
C04416=1012.824,21.215,381.427,-29.088,56.467,-30.850
C04417=1012.823,21.443,381.408,-29.093,56.528,-30.841
C04418=1012.821,21.831,381.378,-29.102,56.634,-30.827
C04419=1012.817,22.160,381.353,-29.108,56.724,-30.812
C04420=1012.815,22.491,381.327,-29.115,56.816,-30.800
C04421=1012.814,22.768,381.306,-29.121,56.891,-30.790
C04422=1012.811,23.132,381.277,-29.129,56.993,-30.776
C04423=1012.807,23.548,381.245,-29.138,57.108,-30.760
C04424=1012.805,23.888,381.218,-29.146,57.204,-30.747
C04425=1012.802,24.267,381.189,-29.154,57.310,-30.732
C04426=1012.799,24.662,381.159,-29.163,57.422,-30.718
C04427=1012.796,25.058,381.128,-29.172,57.535,-30.702
C04428=1012.793,25.454,381.098,-29.181,57.647,-30.689
C04429=1012.790,25.853,381.067,-29.190,57.762,-30.673
C04430=1012.787,26.251,381.035,-29.200,57.876,-30.660
C04431=1012.784,26.647,381.006,-29.209,57.991,-30.645
C04432=1012.781,27.041,380.975,-29.218,58.106,-30.630
C04433=1012.778,27.435,380.944,-29.227,58.221,-30.616
C04434=1012.775,27.828,380.914,-29.236,58.337,-30.602
C04435=1012.772,28.221,380.883,-29.246,58.452,-30.589
C04436=1012.768,28.614,380.853,-29.256,58.570,-30.577
C04437=1012.766,29.009,380.822,-29.265,58.687,-30.563
C04438=1012.763,29.405,380.791,-29.275,58.805,-30.549
C04439=1012.760,29.799,380.761,-29.285,58.924,-30.537
C04440=1012.757,30.195,380.731,-29.295,59.044,-30.524
C04441=1012.754,30.590,380.699,-29.305,59.163,-30.511
C04442=1012.750,30.985,380.669,-29.315,59.283,-30.499
C04443=1012.747,31.381,380.639,-29.325,59.405,-30.486
C04444=1012.745,31.776,380.609,-29.336,59.526,-30.473
C04445=1012.741,32.171,380.578,-29.346,59.648,-30.461
C04446=1012.738,32.567,380.547,-29.357,59.770,-30.450
C04447=1012.735,32.962,380.517,-29.367,59.894,-30.438
C04448=1012.732,33.358,380.485,-29.378,60.016,-30.427
C04449=1012.729,33.752,380.455,-29.389,60.141,-30.416
C04450=1012.726,34.148,380.425,-29.400,60.266,-30.404
C04451=1012.722,34.544,380.394,-29.411,60.391,-30.394
C04452=1012.719,34.938,380.364,-29.422,60.516,-30.383
C04453=1012.716,35.334,380.333,-29.434,60.643,-30.373
C04454=1012.713,35.729,380.302,-29.445,60.768,-30.363
C04455=1012.710,36.125,380.272,-29.457,60.896,-30.352
C04456=1012.707,36.520,380.242,-29.468,61.024,-30.342
C04457=1012.703,36.916,380.211,-29.480,61.151,-30.332
C04458=1012.701,37.311,380.180,-29.492,61.280,-30.324
C04459=1012.698,37.707,380.150,-29.504,61.409,-30.315
C04460=1012.694,38.102,380.119,-29.517,61.538,-30.306
C04461=1012.691,38.497,380.089,-29.529,61.667,-30.298
C04462=1012.688,38.893,380.058,-29.541,61.799,-30.289
C04463=1012.684,39.289,380.028,-29.554,61.929,-30.281
C04464=1012.681,39.683,379.998,-29.567,62.059,-30.274
C04465=1012.678,40.079,379.967,-29.580,62.192,-30.267
C04466=1012.675,40.475,379.937,-29.593,62.324,-30.259
C04467=1012.672,40.870,379.906,-29.606,62.456,-30.252
C04468=1012.669,41.266,379.875,-29.620,62.589,-30.245
C04469=1012.665,41.661,379.845,-29.634,62.722,-30.239
C04470=1012.662,42.057,379.815,-29.648,62.856,-30.234
C04471=1012.659,42.452,379.783,-29.661,62.990,-30.227
C04472=1012.656,42.848,379.754,-29.676,63.125,-30.223
C04473=1012.653,43.244,379.722,-29.690,63.260,-30.216
C04474=1012.649,43.639,379.693,-29.704,63.396,-30.211
C04475=1012.646,44.035,379.662,-29.719,63.531,-30.208
C04476=1012.643,44.431,379.632,-29.734,63.669,-30.203
C04477=1012.640,44.826,379.601,-29.749,63.805,-30.200
C04478=1012.637,45.222,379.570,-29.764,63.943,-30.196
C04479=1012.634,45.618,379.540,-29.780,64.080,-30.194
C04480=1012.630,46.013,379.509,-29.796,64.218,-30.191
C04481=1012.627,46.409,379.479,-29.812,64.358,-30.189
C04482=1012.625,46.805,379.448,-29.828,64.496,-30.187
C04483=1012.621,47.201,379.418,-29.845,64.636,-30.186
C04484=1012.618,47.596,379.388,-29.862,64.776,-30.184
C04485=1012.614,47.992,379.357,-29.879,64.916,-30.183
C04486=1012.611,48.388,379.327,-29.896,65.057,-30.183
C04487=1012.607,48.784,379.296,-29.913,65.198,-30.182
C04488=1012.604,49.180,379.266,-29.931,65.339,-30.184
C04489=1012.601,49.575,379.235,-29.949,65.480,-30.185
C04490=1012.598,49.971,379.205,-29.968,65.624,-30.186
C04491=1012.595,50.366,379.175,-29.987,65.766,-30.188
C04492=1012.592,50.763,379.144,-30.005,65.910,-30.190
C04493=1012.589,51.159,379.114,-30.025,66.054,-30.193
C04494=1012.585,51.554,379.083,-30.044,66.197,-30.195
C04495=1012.582,51.950,379.053,-30.065,66.342,-30.200
C04496=1012.579,52.347,379.023,-30.085,66.486,-30.205
C04497=1012.576,52.742,378.992,-30.105,66.631,-30.209
C04498=1012.573,53.139,378.961,-30.126,66.777,-30.214
C04499=1012.570,53.535,378.931,-30.148,66.923,-30.221
C04500=1012.566,53.931,378.900,-30.169,67.070,-30.226
C04501=1012.563,54.327,378.870,-30.192,67.216,-30.234
C04502=1012.560,54.723,378.840,-30.214,67.363,-30.240
C04503=1012.557,55.118,378.809,-30.237,67.511,-30.248
C04504=1012.554,55.514,378.779,-30.260,67.658,-30.257
C04505=1012.550,55.910,378.749,-30.284,67.808,-30.266
C04506=1012.547,56.306,378.719,-30.308,67.956,-30.277
C04507=1012.545,56.703,378.687,-30.333,68.105,-30.287
C04508=1012.542,57.099,378.658,-30.358,68.254,-30.297
C04509=1012.538,57.495,378.627,-30.383,68.404,-30.310
C04510=1012.535,57.890,378.596,-30.409,68.554,-30.321
C04511=1012.532,58.286,378.567,-30.436,68.705,-30.335
C04512=1012.528,58.683,378.536,-30.463,68.857,-30.349
C04513=1012.525,59.079,378.506,-30.491,69.008,-30.363
C04514=1012.523,59.475,378.475,-30.519,69.159,-30.379
C04515=1012.520,59.871,378.445,-30.547,69.311,-30.394
C04516=1012.516,60.267,378.414,-30.577,69.463,-30.412
C04517=1012.513,60.663,378.384,-30.607,69.616,-30.429
C04518=1012.510,61.058,378.354,-30.637,69.770,-30.447
C04519=1012.507,61.455,378.323,-30.669,69.923,-30.467
C04520=1012.504,61.851,378.293,-30.700,70.077,-30.486
C04521=1012.501,62.250,378.263,-30.733,70.231,-30.507
C04522=1012.499,62.533,378.241,-30.757,70.342,-30.523
C04523=1012.497,62.752,378.224,-30.776,70.428,-30.536
C04524=1012.495,62.994,378.205,-30.796,70.523,-30.549
C04525=1012.493,63.243,378.186,-30.818,70.620,-30.564
C04526=1012.492,63.478,378.168,-30.838,70.712,-30.577
C04527=1012.489,63.689,378.152,-30.857,70.795,-30.590
C04528=1012.488,64.095,378.116,-30.866,70.841,-30.596
C04529=1012.488,64.314,378.096,-30.868,70.847,-30.596
C04530=1012.486,64.540,378.075,-30.868,70.852,-30.595
C04531=1012.487,64.766,378.053,-30.867,70.858,-30.593
C04532=1012.486,64.989,378.033,-30.869,70.863,-30.593
C04533=1012.485,65.208,378.012,-30.869,70.868,-30.592
C04534=1012.485,65.423,377.992,-30.869,70.873,-30.592
C04535=1012.484,65.631,377.973,-30.870,70.878,-30.591
C04536=1012.483,66.024,377.936,-30.871,70.887,-30.591
C04537=1012.482,66.351,377.906,-30.871,70.895,-30.589
C04538=1012.481,66.715,377.871,-30.872,70.904,-30.588
C04539=1012.480,67.112,377.834,-30.872,70.914,-30.586
C04540=1012.478,67.510,377.797,-30.874,70.922,-30.586
C04541=1012.477,67.912,377.759,-30.874,70.932,-30.584
C04542=1012.476,68.323,377.721,-30.876,70.943,-30.584
C04543=1012.475,68.740,377.682,-30.876,70.953,-30.582
C04544=1012.474,69.157,377.643,-30.878,70.963,-30.582
C04545=1012.473,69.564,377.605,-30.878,70.973,-30.580
C04546=1012.471,69.969,377.567,-30.879,70.983,-30.578
C04547=1012.471,70.373,377.528,-30.880,70.992,-30.578
C04548=1012.469,70.778,377.490,-30.882,71.003,-30.578
C04549=1012.468,71.182,377.452,-30.882,71.013,-30.576
C04550=1012.467,71.586,377.414,-30.883,71.022,-30.575
C04551=1012.465,71.991,377.376,-30.884,71.033,-30.574
C04552=1012.464,72.398,377.337,-30.885,71.043,-30.573
C04553=1012.463,72.805,377.299,-30.886,71.053,-30.572
C04554=1012.462,73.215,377.261,-30.887,71.063,-30.570
C04555=1012.461,73.627,377.222,-30.888,71.074,-30.570
C04556=1012.460,74.041,377.183,-30.890,71.085,-30.570
C04557=1012.459,74.260,377.162,-30.890,71.089,-30.569
C04558=1012.458,74.489,377.140,-30.891,71.096,-30.568
C04559=1012.457,74.715,377.119,-30.892,71.102,-30.568
C04560=1012.457,74.931,377.099,-30.892,71.107,-30.568
C04561=1012.456,75.139,377.079,-30.893,71.112,-30.568
C04562=1012.456,75.554,377.040,-30.894,71.122,-30.566
C04563=1012.454,75.962,377.002,-30.894,71.134,-30.564
C04564=1012.452,76.364,376.963,-30.897,71.143,-30.566
C04565=1012.451,76.758,376.926,-30.897,71.153,-30.564
C04566=1012.450,77.145,376.890,-30.899,71.164,-30.564
C04567=1012.449,77.527,376.853,-30.899,71.174,-30.562
C04568=1012.447,77.909,376.817,-30.900,71.183,-30.560
C04569=1012.447,78.292,376.781,-30.902,71.193,-30.562
C04570=1012.445,78.681,376.744,-30.903,71.203,-30.560
C04571=1012.444,79.075,376.706,-30.904,71.214,-30.560
C04572=1012.443,79.477,376.668,-30.906,71.224,-30.560
C04573=1012.441,79.886,376.629,-30.906,71.236,-30.558
C04574=1012.440,80.298,376.590,-30.908,71.246,-30.557
C04575=1012.439,80.681,376.554,-30.909,71.257,-30.557
C04576=1012.438,81.045,376.519,-30.911,71.266,-30.557
C04577=1012.437,81.438,376.481,-30.912,71.276,-30.557
C04578=1012.435,81.854,376.442,-30.913,71.288,-30.555
C04579=1012.434,82.267,376.402,-30.914,71.299,-30.555
C04580=1012.433,82.680,376.363,-30.916,71.309,-30.554
C04581=1012.431,83.092,376.324,-30.916,71.321,-30.552
C04582=1012.430,83.503,376.285,-30.919,71.332,-30.554
C04583=1012.429,83.912,376.246,-30.920,71.343,-30.553
C04584=1012.427,84.321,376.206,-30.921,71.354,-30.551
C04585=1012.426,84.728,376.168,-30.922,71.365,-30.551
C04586=1012.425,85.133,376.129,-30.925,71.376,-30.552
C04587=1012.423,85.537,376.090,-30.925,71.388,-30.550
C04588=1012.422,85.940,376.052,-30.927,71.398,-30.550
C04589=1012.421,86.343,376.013,-30.928,71.409,-30.550
C04590=1012.419,86.743,375.975,-30.931,71.420,-30.551
C04591=1012.418,87.142,375.936,-30.931,71.432,-30.549
C04592=1012.417,87.537,375.899,-30.933,71.442,-30.549
C04593=1012.415,87.921,375.862,-30.934,71.453,-30.549
C04594=1012.414,88.298,375.825,-30.936,71.463,-30.548
C04595=1012.413,88.673,375.790,-30.937,71.474,-30.548
C04596=1012.412,89.052,375.753,-30.939,71.485,-30.548
C04597=1012.410,89.436,375.717,-30.940,71.495,-30.548
C04598=1012.409,89.832,375.679,-30.942,71.506,-30.548
C04599=1012.408,90.067,375.655,-30.942,71.512,-30.546
C04600=1012.407,90.341,375.629,-30.943,71.520,-30.547
C04601=1012.406,90.621,375.602,-30.945,71.527,-30.547
C04602=1012.406,90.867,375.579,-30.946,71.534,-30.547
C04603=1012.404,91.269,375.540,-30.947,71.545,-30.547
C04604=1012.403,91.664,375.502,-30.949,71.557,-30.547
C04605=1012.401,92.059,375.464,-30.951,71.569,-30.546
C04606=1012.400,92.453,375.426,-30.953,71.581,-30.548
C04607=1012.399,92.848,375.388,-30.954,71.592,-30.546
C04608=1012.397,93.243,375.350,-30.956,71.603,-30.547
C04609=1012.396,93.637,375.311,-30.958,71.614,-30.547
C04610=1012.395,94.032,375.273,-30.959,71.625,-30.547
C04611=1012.393,94.426,375.236,-30.961,71.635,-30.546
C04612=1012.392,94.820,375.197,-30.962,71.646,-30.546
C04613=1012.390,95.215,375.159,-30.964,71.658,-30.546
C04614=1012.389,95.610,375.121,-30.966,71.669,-30.547
C04615=1012.388,96.004,375.082,-30.968,71.682,-30.547
C04616=1012.387,96.399,375.045,-30.970,71.694,-30.548
C04617=1012.385,96.794,375.006,-30.972,71.707,-30.547
C04618=1012.384,97.188,374.968,-30.973,71.717,-30.547
C04619=1012.383,97.582,374.930,-30.975,71.728,-30.547
C04620=1012.381,97.977,374.891,-30.977,71.739,-30.548
C04621=1012.380,98.371,374.853,-30.980,71.751,-30.549
C04622=1012.379,98.766,374.815,-30.981,71.763,-30.549
C04623=1012.377,99.160,374.776,-30.983,71.775,-30.549
C04624=1012.376,99.555,374.739,-30.986,71.788,-30.550
C04625=1012.374,99.948,374.700,-30.988,71.801,-30.551
C04626=1012.372,100.343,374.662,-30.990,71.812,-30.551
C04627=1012.371,100.737,374.624,-30.991,71.822,-30.551
C04628=1012.370,101.132,374.585,-30.993,71.834,-30.550
C04629=1012.368,101.526,374.547,-30.995,71.846,-30.551
C04630=1012.367,101.920,374.508,-30.997,71.858,-30.551
C04631=1012.365,102.315,374.470,-30.999,71.871,-30.552
C04632=1012.364,102.709,374.431,-31.001,71.883,-30.552
C04633=1012.363,103.104,374.392,-31.005,71.897,-30.554
C04634=1012.361,103.498,374.355,-31.006,71.907,-30.554
C04635=1012.361,103.892,374.316,-31.008,71.920,-30.554
C04636=1012.359,104.287,374.277,-31.009,71.930,-30.554
C04637=1012.357,104.681,374.240,-31.011,71.942,-30.553
C04638=1012.355,105.075,374.200,-31.014,71.954,-30.556
C04639=1012.354,105.469,374.162,-31.017,71.967,-30.557
C04640=1012.352,105.864,374.124,-31.019,71.980,-30.559
C04641=1012.351,106.258,374.085,-31.021,71.994,-30.558
C04642=1012.350,106.652,374.046,-31.024,72.006,-30.559
C04643=1012.349,107.046,374.008,-31.025,72.018,-30.559
C04644=1012.347,107.441,373.968,-31.028,72.029,-30.560
C04645=1012.346,107.835,373.931,-31.030,72.041,-30.560
C04646=1012.344,108.230,373.892,-31.032,72.053,-30.562
C04647=1012.343,108.623,373.854,-31.035,72.066,-30.563
C04648=1012.341,109.017,373.814,-31.036,72.079,-30.562
C04649=1012.340,109.411,373.776,-31.040,72.093,-30.565
C04650=1012.338,109.806,373.737,-31.043,72.106,-30.566
C04651=1012.337,110.200,373.698,-31.045,72.117,-30.567
C04652=1012.336,110.595,373.660,-31.047,72.130,-30.567
C04653=1012.334,110.989,373.621,-31.049,72.141,-30.569
C04654=1012.333,111.383,373.582,-31.052,72.154,-30.570
C04655=1012.331,111.777,373.543,-31.055,72.167,-30.571
C04656=1012.330,112.172,373.504,-31.057,72.180,-30.572
C04657=1012.329,112.566,373.466,-31.059,72.194,-30.572
C04658=1012.327,112.960,373.427,-31.063,72.207,-30.574
C04659=1012.325,113.354,373.389,-31.064,72.220,-30.574
C04660=1012.324,113.748,373.349,-31.067,72.231,-30.576
C04661=1012.322,114.142,373.310,-31.069,72.244,-30.577
C04662=1012.321,114.536,373.272,-31.072,72.257,-30.578
C04663=1012.319,114.931,373.233,-31.075,72.270,-30.579
C04664=1012.318,115.325,373.194,-31.077,72.283,-30.581
C04665=1012.316,115.719,373.155,-31.081,72.296,-30.583
C04666=1012.315,116.113,373.116,-31.084,72.311,-30.584
C04667=1012.313,116.508,373.077,-31.086,72.323,-30.584
C04668=1012.312,116.902,373.038,-31.089,72.335,-30.587
C04669=1012.311,117.295,372.999,-31.091,72.347,-30.587
C04670=1012.309,117.690,372.960,-31.093,72.360,-30.588
C04671=1012.308,118.084,372.921,-31.096,72.373,-30.590
C04672=1012.306,118.478,372.882,-31.100,72.387,-30.592
C04673=1012.304,118.873,372.842,-31.103,72.402,-30.593
C04674=1012.303,119.267,372.804,-31.106,72.415,-30.596
C04675=1012.302,119.661,372.765,-31.108,72.429,-30.596
C04676=1012.300,120.055,372.726,-31.112,72.441,-30.599
C04677=1012.299,120.449,372.686,-31.114,72.454,-30.600
C04678=1012.297,120.844,372.647,-31.117,72.467,-30.602
C04679=1012.295,121.238,372.608,-31.120,72.480,-30.603
C04680=1012.294,121.632,372.569,-31.123,72.494,-30.606
C04681=1012.293,122.026,372.530,-31.126,72.508,-30.607
C04682=1012.291,122.420,372.490,-31.129,72.523,-30.608
C04683=1012.290,122.814,372.451,-31.133,72.536,-30.611
C04684=1012.288,123.209,372.412,-31.136,72.549,-30.612
C04685=1012.286,123.603,372.373,-31.138,72.562,-30.614
C04686=1012.286,123.997,372.333,-31.141,72.575,-30.615
C04687=1012.284,124.392,372.294,-31.144,72.588,-30.617
C04688=1012.282,124.786,372.255,-31.148,72.602,-30.619
C04689=1012.281,125.180,372.215,-31.151,72.616,-30.621
C04690=1012.279,125.574,372.176,-31.154,72.630,-30.624
C04691=1012.278,125.968,372.138,-31.158,72.645,-30.626
C04692=1012.277,126.363,372.098,-31.161,72.658,-30.628
C04693=1012.275,126.756,372.059,-31.164,72.671,-30.629
C04694=1012.273,127.152,372.019,-31.167,72.685,-30.632
C04695=1012.272,127.546,371.980,-31.170,72.698,-30.634
C04696=1012.270,127.940,371.940,-31.174,72.712,-30.637
C04697=1012.269,128.334,371.901,-31.177,72.726,-30.638
C04698=1012.267,128.728,371.862,-31.181,72.742,-30.641
C04699=1012.266,129.122,371.822,-31.185,72.757,-30.643
C04700=1012.264,129.517,371.782,-31.189,72.770,-30.646
C04701=1012.263,129.911,371.742,-31.191,72.783,-30.648
C04702=1012.261,130.305,371.703,-31.194,72.796,-30.649
C04703=1012.260,130.700,371.664,-31.198,72.810,-30.652
C04704=1012.259,131.094,371.624,-31.202,72.824,-30.656
C04705=1012.257,131.488,371.585,-31.205,72.838,-30.657
C04706=1012.256,131.882,371.545,-31.209,72.854,-30.660
C04707=1012.254,132.277,371.506,-31.213,72.869,-30.663
C04708=1012.252,132.672,371.466,-31.217,72.884,-30.665
C04709=1012.251,133.065,371.426,-31.220,72.897,-30.667
C04710=1012.249,133.460,371.387,-31.224,72.911,-30.670
C04711=1012.249,133.854,371.347,-31.227,72.924,-30.673
C04712=1012.246,134.249,371.307,-31.231,72.938,-30.676
C04713=1012.245,134.644,371.268,-31.234,72.953,-30.678
C04714=1012.244,134.874,371.245,-31.237,72.962,-30.680
C04715=1012.243,135.133,371.219,-31.240,72.972,-30.682
C04716=1012.242,135.544,371.177,-31.244,72.987,-30.685
C04717=1012.240,135.913,371.140,-31.249,73.002,-30.689
C04718=1012.239,136.253,371.106,-31.251,73.015,-30.691
C04719=1012.238,136.574,371.073,-31.254,73.026,-30.693
C04720=1012.236,136.895,371.041,-31.258,73.038,-30.696
C04721=1012.235,137.238,371.007,-31.261,73.051,-30.698
C04722=1012.234,137.587,370.971,-31.265,73.063,-30.701
C04723=1012.233,137.887,370.941,-31.268,73.074,-30.703
C04724=1012.231,138.283,370.900,-31.272,73.089,-30.706
C04725=1012.230,138.502,370.878,-31.274,73.097,-30.709
C04726=1012.229,138.738,370.855,-31.276,73.106,-30.709
C04727=1012.229,138.987,370.830,-31.279,73.116,-30.711
C04728=1012.227,139.244,370.804,-31.282,73.125,-30.715
C04729=1012.227,139.507,370.777,-31.284,73.135,-30.715
C04730=1012.226,139.768,370.751,-31.287,73.145,-30.717
C04731=1012.225,140.021,370.725,-31.289,73.154,-30.720
C04732=1012.224,140.263,370.701,-31.292,73.162,-30.722
C04733=1012.224,140.491,370.678,-31.294,73.171,-30.722
C04734=1012.222,140.702,370.657,-31.296,73.179,-30.725
C04735=1012.221,140.920,370.634,-31.299,73.187,-30.727
C04736=1012.220,141.324,370.594,-31.303,73.203,-30.730
C04737=1012.218,141.590,370.567,-31.306,73.212,-30.732
C04738=1012.219,141.790,370.546,-31.308,73.220,-30.735
C04739=1012.217,142.191,370.506,-31.312,73.236,-30.738
C04740=1012.215,142.591,370.465,-31.317,73.251,-30.741
C04741=1012.214,142.993,370.424,-31.322,73.265,-30.746
C04742=1012.212,143.396,370.383,-31.326,73.281,-30.749
C04743=1012.211,143.799,370.342,-31.331,73.297,-30.754
C04744=1012.209,144.204,370.301,-31.335,73.312,-30.757
C04745=1012.208,144.608,370.260,-31.340,73.327,-30.760
C04746=1012.206,145.012,370.220,-31.344,73.342,-30.763
C04747=1012.205,145.418,370.178,-31.349,73.358,-30.768
C04748=1012.203,145.824,370.137,-31.353,73.374,-30.771
C04749=1012.202,146.229,370.095,-31.359,73.390,-30.776
C04750=1012.200,146.635,370.055,-31.363,73.405,-30.779
C04751=1012.199,147.044,370.013,-31.368,73.421,-30.784
C04752=1012.348,146.999,369.573,-29.484,63.365,-29.613
C04753=1012.350,146.590,369.614,-29.482,63.348,-29.614
C04754=1012.352,146.184,369.656,-29.481,63.332,-29.616
C04755=1012.353,145.779,369.697,-29.480,63.316,-29.618
C04756=1012.354,145.373,369.738,-29.478,63.300,-29.618
C04757=1012.356,144.967,369.780,-29.477,63.284,-29.619
C04758=1012.357,144.563,369.820,-29.476,63.267,-29.622
C04759=1012.360,144.158,369.862,-29.475,63.252,-29.623
C04760=1012.361,143.755,369.902,-29.474,63.236,-29.624
C04761=1012.363,143.351,369.943,-29.472,63.220,-29.625
C04762=1012.364,142.949,369.984,-29.471,63.205,-29.627
C04763=1012.366,142.547,370.026,-29.470,63.189,-29.628
C04764=1012.367,142.145,370.066,-29.469,63.173,-29.629
C04765=1012.369,141.745,370.107,-29.467,63.157,-29.630
C04766=1012.369,141.545,370.127,-29.467,63.150,-29.631
C04767=1012.371,141.280,370.154,-29.466,63.139,-29.634
C04768=1012.373,140.874,370.195,-29.465,63.123,-29.635
C04769=1012.373,140.657,370.217,-29.464,63.115,-29.635
C04770=1012.374,140.445,370.238,-29.463,63.107,-29.635
C04771=1012.375,140.219,370.261,-29.463,63.098,-29.637
C04772=1012.376,139.976,370.286,-29.463,63.089,-29.638
C04773=1012.377,139.723,370.311,-29.462,63.079,-29.639
C04774=1012.378,139.462,370.338,-29.461,63.069,-29.640
C04775=1012.379,139.200,370.364,-29.460,63.059,-29.640
C04776=1012.380,138.942,370.391,-29.459,63.049,-29.641
C04777=1012.381,138.693,370.415,-29.459,63.040,-29.643
C04778=1012.382,138.457,370.439,-29.458,63.030,-29.643
C04779=1012.383,138.239,370.461,-29.458,63.023,-29.644
C04780=1012.384,137.843,370.502,-29.456,63.007,-29.646
C04781=1012.386,137.542,370.532,-29.455,62.995,-29.647
C04782=1012.387,137.194,370.567,-29.455,62.982,-29.649
C04783=1012.389,136.851,370.602,-29.454,62.969,-29.650
C04784=1012.390,136.529,370.634,-29.453,62.957,-29.652
C04785=1012.391,136.209,370.667,-29.452,62.944,-29.653
C04786=1012.392,135.868,370.701,-29.451,62.932,-29.654
C04787=1012.394,135.499,370.738,-29.450,62.917,-29.656
C04788=1012.396,135.089,370.779,-29.449,62.900,-29.659
C04789=1012.397,134.830,370.805,-29.448,62.890,-29.659
C04790=1012.398,134.599,370.829,-29.447,62.882,-29.659
C04791=1012.399,134.204,370.868,-29.446,62.866,-29.661
C04792=1012.401,133.810,370.908,-29.445,62.851,-29.663
C04793=1012.402,133.415,370.948,-29.445,62.836,-29.665
C04794=1012.404,133.021,370.987,-29.444,62.823,-29.667
C04795=1012.405,132.627,371.027,-29.443,62.810,-29.669
C04796=1012.407,132.233,371.066,-29.442,62.794,-29.670
C04797=1012.409,131.838,371.107,-29.440,62.779,-29.671
C04798=1012.410,131.444,371.146,-29.440,62.764,-29.674
C04799=1012.412,131.049,371.185,-29.439,62.749,-29.676
C04800=1012.413,130.656,371.225,-29.438,62.734,-29.678
C04801=1012.416,130.261,371.265,-29.437,62.720,-29.679
C04802=1012.417,129.867,371.305,-29.436,62.706,-29.681
C04803=1012.418,129.472,371.344,-29.435,62.693,-29.683
C04804=1012.420,129.078,371.383,-29.434,62.678,-29.685
C04805=1012.421,128.684,371.423,-29.433,62.663,-29.687
C04806=1012.423,128.290,371.462,-29.432,62.648,-29.689
C04807=1012.425,127.896,371.501,-29.431,62.633,-29.691
C04808=1012.427,127.502,371.541,-29.431,62.619,-29.694
C04809=1012.428,127.107,371.580,-29.430,62.605,-29.695
C04810=1012.429,126.713,371.621,-29.429,62.591,-29.697
C04811=1012.431,126.318,371.660,-29.428,62.578,-29.699
C04812=1012.433,125.924,371.699,-29.427,62.565,-29.700
C04813=1012.434,125.530,371.739,-29.427,62.549,-29.704
C04814=1012.436,125.136,371.778,-29.425,62.535,-29.705
C04815=1012.437,124.742,371.817,-29.425,62.520,-29.707
C04816=1012.439,124.347,371.856,-29.424,62.505,-29.710
C04817=1012.440,123.954,371.896,-29.423,62.492,-29.711
C04818=1012.442,123.559,371.935,-29.422,62.479,-29.713
C04819=1012.444,123.165,371.974,-29.421,62.465,-29.715
C04820=1012.445,122.771,372.013,-29.421,62.453,-29.718
C04821=1012.447,122.377,372.053,-29.420,62.437,-29.719
C04822=1012.448,121.983,372.092,-29.419,62.422,-29.721
C04823=1012.450,121.588,372.131,-29.418,62.408,-29.725
C04824=1012.452,121.194,372.170,-29.417,62.394,-29.726
C04825=1012.453,120.800,372.209,-29.417,62.380,-29.729
C04826=1012.455,120.406,372.249,-29.416,62.367,-29.731
C04827=1012.457,120.011,372.288,-29.416,62.354,-29.734
C04828=1012.458,119.617,372.327,-29.415,62.341,-29.735
C04829=1012.459,119.223,372.365,-29.414,62.328,-29.737
C04830=1012.461,118.829,372.405,-29.413,62.313,-29.740
C04831=1012.462,118.435,372.444,-29.412,62.298,-29.742
C04832=1012.464,118.041,372.483,-29.411,62.285,-29.744
C04833=1012.466,117.646,372.522,-29.411,62.270,-29.747
C04834=1012.468,117.253,372.561,-29.410,62.257,-29.749
C04835=1012.469,116.859,372.600,-29.410,62.245,-29.752
C04836=1012.470,116.464,372.639,-29.409,62.233,-29.753
C04837=1012.472,116.070,372.678,-29.408,62.220,-29.755
C04838=1012.474,115.676,372.717,-29.407,62.205,-29.757
C04839=1012.475,115.281,372.756,-29.407,62.191,-29.761
C04840=1012.476,114.887,372.795,-29.406,62.177,-29.764
C04841=1012.478,114.493,372.834,-29.406,62.163,-29.766
C04842=1012.480,114.099,372.873,-29.405,62.150,-29.768
C04843=1012.481,113.704,372.912,-29.404,62.138,-29.770
C04844=1012.483,113.311,372.950,-29.404,62.125,-29.773
C04845=1012.484,112.917,372.990,-29.403,62.113,-29.775
C04846=1012.486,112.522,373.028,-29.402,62.099,-29.777
C04847=1012.488,112.128,373.067,-29.402,62.084,-29.780
C04848=1012.489,111.734,373.106,-29.401,62.071,-29.782
C04849=1012.491,111.340,373.145,-29.400,62.058,-29.784
C04850=1012.492,110.945,373.184,-29.400,62.045,-29.787
C04851=1012.493,110.551,373.222,-29.399,62.032,-29.789
C04852=1012.496,110.158,373.261,-29.399,62.020,-29.792
C04853=1012.497,109.763,373.300,-29.398,62.009,-29.794
C04854=1012.498,109.369,373.339,-29.398,61.995,-29.797
C04855=1012.500,108.975,373.378,-29.397,61.981,-29.800
C04856=1012.501,108.581,373.416,-29.397,61.967,-29.802
C04857=1012.503,108.186,373.454,-29.396,61.954,-29.804
C04858=1012.504,107.791,373.494,-29.395,61.942,-29.807
C04859=1012.506,107.398,373.532,-29.395,61.929,-29.810
C04860=1012.508,107.004,373.571,-29.395,61.917,-29.813
C04861=1012.509,106.610,373.609,-29.394,61.906,-29.815
C04862=1012.511,106.215,373.648,-29.394,61.893,-29.818
C04863=1012.512,105.820,373.687,-29.393,61.878,-29.820
C04864=1012.513,105.426,373.725,-29.392,61.866,-29.823
C04865=1012.515,105.033,373.764,-29.392,61.853,-29.825
C04866=1012.517,104.638,373.802,-29.391,61.840,-29.828
C04867=1012.518,104.244,373.841,-29.391,61.828,-29.831
C04868=1012.519,103.850,373.879,-29.390,61.815,-29.833
C04869=1012.521,103.455,373.918,-29.390,61.804,-29.836
C04870=1012.522,103.061,373.956,-29.390,61.793,-29.839
C04871=1012.524,102.666,373.995,-29.389,61.779,-29.841
C04872=1012.526,102.273,374.033,-29.389,61.765,-29.845
C04873=1012.527,101.878,374.072,-29.388,61.752,-29.847
C04874=1012.528,101.484,374.110,-29.387,61.739,-29.850
C04875=1012.530,101.089,374.149,-29.387,61.728,-29.853
C04876=1012.531,100.695,374.187,-29.387,61.716,-29.855
C04877=1012.533,100.300,374.225,-29.387,61.705,-29.858
C04878=1012.534,99.906,374.264,-29.386,61.694,-29.861
C04879=1012.536,99.511,374.302,-29.386,61.681,-29.864
C04880=1012.538,99.118,374.340,-29.385,61.668,-29.866
C04881=1012.539,98.723,374.378,-29.385,61.655,-29.870
C04882=1012.541,98.329,374.417,-29.384,61.642,-29.873
C04883=1012.542,97.934,374.455,-29.384,61.631,-29.874
C04884=1012.543,97.540,374.494,-29.384,61.619,-29.878
C04885=1012.545,97.145,374.532,-29.383,61.608,-29.880
C04886=1012.546,96.751,374.570,-29.383,61.597,-29.882
C04887=1012.547,96.357,374.608,-29.382,61.585,-29.885
C04888=1012.549,95.962,374.647,-29.382,61.572,-29.888
C04889=1012.551,95.568,374.685,-29.381,61.558,-29.892
C04890=1012.552,95.174,374.722,-29.381,61.546,-29.895
C04891=1012.554,94.779,374.761,-29.381,61.535,-29.897
C04892=1012.555,94.385,374.799,-29.381,61.523,-29.901
C04893=1012.556,93.990,374.837,-29.380,61.512,-29.903
C04894=1012.558,93.595,374.875,-29.380,61.501,-29.905
C04895=1012.559,93.200,374.913,-29.380,61.491,-29.908
C04896=1012.560,92.806,374.952,-29.379,61.479,-29.911
C04897=1012.562,92.411,374.990,-29.379,61.467,-29.915
C04898=1012.563,92.017,375.028,-29.379,61.455,-29.918
C04899=1012.565,91.622,375.066,-29.378,61.442,-29.921
C04900=1012.566,91.227,375.103,-29.378,61.430,-29.924
C04901=1012.568,90.825,375.143,-29.377,61.419,-29.926
C04902=1012.569,90.579,375.166,-29.378,61.411,-29.930
C04903=1012.570,90.300,375.193,-29.377,61.404,-29.931
C04904=1012.570,90.025,375.219,-29.377,61.396,-29.932
C04905=1012.572,89.790,375.243,-29.377,61.391,-29.933
C04906=1012.573,89.395,375.281,-29.377,61.379,-29.937
C04907=1012.574,89.010,375.318,-29.376,61.368,-29.939
C04908=1012.576,88.631,375.354,-29.376,61.357,-29.944
C04909=1012.577,88.256,375.389,-29.376,61.346,-29.946
C04910=1012.578,87.879,375.426,-29.376,61.336,-29.948
C04911=1012.580,87.494,375.464,-29.376,61.324,-29.952
C04912=1012.581,87.101,375.500,-29.375,61.313,-29.955
C04913=1012.582,86.702,375.539,-29.375,61.301,-29.958
C04914=1012.584,86.300,375.578,-29.375,61.291,-29.961
C04915=1012.585,85.899,375.615,-29.375,61.279,-29.965
C04916=1012.587,85.496,375.655,-29.374,61.268,-29.967
C04917=1012.588,85.092,375.693,-29.374,61.256,-29.971
C04918=1012.589,84.686,375.732,-29.374,61.246,-29.973
C04919=1012.590,84.279,375.771,-29.374,61.234,-29.977
C04920=1012.592,83.870,375.810,-29.374,61.222,-29.981
C04921=1012.593,83.461,375.849,-29.373,61.211,-29.983
C04922=1012.594,83.050,375.889,-29.373,61.199,-29.986
C04923=1012.597,82.639,375.928,-29.373,61.187,-29.990
C04924=1012.597,82.226,375.967,-29.372,61.176,-29.992
C04925=1012.599,81.812,376.007,-29.372,61.165,-29.996
C04926=1012.600,81.397,376.046,-29.372,61.153,-30.000
C04927=1012.602,81.003,376.084,-29.372,61.143,-30.003
C04928=1012.603,80.639,376.118,-29.372,61.133,-30.006
C04929=1012.604,80.257,376.155,-29.372,61.122,-30.009
C04930=1012.605,79.845,376.194,-29.371,61.111,-30.011
C04931=1012.607,79.436,376.233,-29.371,61.100,-30.016
C04932=1012.609,79.034,376.271,-29.371,61.090,-30.018
C04933=1012.610,78.639,376.309,-29.371,61.080,-30.021
C04934=1012.610,78.250,376.345,-29.371,61.068,-30.025
C04935=1012.612,77.867,376.382,-29.371,61.058,-30.029
C04936=1012.614,77.486,376.418,-29.371,61.048,-30.032
C04937=1012.614,77.103,376.454,-29.370,61.037,-30.034
C04938=1012.616,76.716,376.491,-29.370,61.027,-30.037
C04939=1012.617,76.323,376.528,-29.370,61.017,-30.041
C04940=1012.619,75.921,376.566,-29.370,61.006,-30.043
C04941=1012.620,75.513,376.605,-29.370,60.995,-30.048
C04942=1012.621,75.098,376.644,-29.370,60.984,-30.050
C04943=1012.622,74.889,376.663,-29.370,60.979,-30.052
C04944=1012.622,74.674,376.685,-29.370,60.973,-30.055
C04945=1012.623,74.448,376.706,-29.369,60.968,-30.056
C04946=1012.624,74.220,376.727,-29.369,60.961,-30.058
C04947=1012.625,74.001,376.748,-29.369,60.956,-30.059
C04948=1012.626,73.586,376.787,-29.370,60.945,-30.064
C04949=1012.627,73.173,376.826,-29.369,60.934,-30.067
C04950=1012.629,72.764,376.864,-29.369,60.924,-30.070
C04951=1012.630,72.357,376.903,-29.369,60.913,-30.074
C04952=1012.631,71.951,376.941,-29.369,60.902,-30.077
C04953=1012.632,71.546,376.979,-29.369,60.892,-30.080
C04954=1012.634,71.141,377.018,-29.369,60.882,-30.084
C04955=1012.635,70.737,377.056,-29.369,60.871,-30.087
C04956=1012.636,70.332,377.094,-29.369,60.861,-30.091
C04957=1012.637,69.928,377.131,-29.369,60.851,-30.094
C04958=1012.639,69.523,377.170,-29.369,60.841,-30.097
C04959=1012.640,69.115,377.208,-29.369,60.831,-30.101
C04960=1012.641,68.700,377.247,-29.368,60.821,-30.104
C04961=1012.643,68.282,377.286,-29.369,60.810,-30.109
C04962=1012.643,67.871,377.324,-29.369,60.800,-30.112
C04963=1012.644,67.469,377.362,-29.369,60.790,-30.115
C04964=1012.646,67.072,377.400,-29.369,60.780,-30.118
C04965=1012.647,66.674,377.437,-29.368,60.770,-30.122
C04966=1012.648,66.310,377.471,-29.368,60.761,-30.125
C04967=1012.649,65.983,377.502,-29.368,60.753,-30.127
C04968=1012.651,65.590,377.538,-29.369,60.744,-30.131
C04969=1012.651,65.382,377.557,-29.369,60.739,-30.133
C04970=1012.651,65.168,377.578,-29.368,60.733,-30.134
C04971=1012.652,64.949,377.598,-29.369,60.727,-30.137
C04972=1012.652,64.726,377.619,-29.368,60.722,-30.139
C04973=1012.654,64.500,377.640,-29.368,60.717,-30.140
C04974=1012.654,64.273,377.661,-29.369,60.711,-30.143
C04975=1012.654,64.054,377.682,-29.369,60.706,-30.145
C04976=1012.657,63.649,377.718,-29.365,60.655,-30.150
C04977=1012.659,63.438,377.734,-29.357,60.568,-30.157
C04978=1012.662,63.202,377.752,-29.348,60.469,-30.165
C04979=1012.664,62.954,377.772,-29.339,60.366,-30.172
C04980=1012.666,62.712,377.790,-29.330,60.266,-30.179
C04981=1012.669,62.492,377.807,-29.322,60.175,-30.186
C04982=1012.672,62.210,377.829,-29.312,60.057,-30.195
C04983=1012.676,61.810,377.859,-29.298,59.892,-30.210
C04984=1012.681,61.415,377.891,-29.283,59.730,-30.223
C04985=1012.685,61.019,377.921,-29.270,59.567,-30.238
C04986=1012.689,60.623,377.951,-29.256,59.405,-30.252
C04987=1012.693,60.227,377.982,-29.242,59.243,-30.267
C04988=1012.697,59.830,378.013,-29.229,59.081,-30.282
C04989=1012.702,59.435,378.043,-29.216,58.920,-30.299
C04990=1012.706,59.038,378.074,-29.202,58.759,-30.315
C04991=1012.710,58.643,378.104,-29.189,58.599,-30.331
C04992=1012.714,58.246,378.135,-29.176,58.439,-30.348
C04993=1012.719,57.851,378.165,-29.163,58.280,-30.365
C04994=1012.722,57.455,378.196,-29.151,58.121,-30.383
C04995=1012.727,57.059,378.227,-29.138,57.963,-30.400
C04996=1012.731,56.663,378.258,-29.125,57.804,-30.418
C04997=1012.736,56.267,378.288,-29.113,57.646,-30.436
C04998=1012.740,55.871,378.319,-29.100,57.489,-30.454
C04999=1012.744,55.475,378.349,-29.088,57.332,-30.474
C05000=1012.748,55.079,378.379,-29.076,57.176,-30.492
C05001=1012.753,54.683,378.411,-29.063,57.020,-30.511
C05002=1012.757,54.287,378.441,-29.052,56.865,-30.532
C05003=1012.761,53.892,378.471,-29.040,56.710,-30.552
C05004=1012.765,53.495,378.502,-29.028,56.556,-30.571
C05005=1012.770,53.099,378.533,-29.016,56.401,-30.592
C05006=1012.774,52.703,378.564,-29.004,56.247,-30.612
C05007=1012.778,52.308,378.594,-28.992,56.093,-30.634
C05008=1012.782,51.912,378.625,-28.980,55.941,-30.654
C05009=1012.787,51.516,378.656,-28.969,55.789,-30.676
C05010=1012.791,51.119,378.686,-28.958,55.637,-30.698
C05011=1012.795,50.724,378.717,-28.946,55.485,-30.719
C05012=1012.799,50.328,378.748,-28.934,55.334,-30.741
C05013=1012.803,49.932,378.778,-28.923,55.184,-30.764
C05014=1012.808,49.536,378.810,-28.912,55.034,-30.787
C05015=1012.812,49.141,378.840,-28.901,54.883,-30.810
C05016=1012.816,48.744,378.871,-28.889,54.735,-30.833
C05017=1012.820,48.349,378.902,-28.878,54.586,-30.856
C05018=1012.825,47.954,378.932,-28.867,54.438,-30.879
C05019=1012.828,47.557,378.963,-28.856,54.290,-30.904
C05020=1012.833,47.162,378.994,-28.845,54.143,-30.927
C05021=1012.837,46.766,379.024,-28.834,53.996,-30.952
C05022=1012.841,46.371,379.055,-28.823,53.849,-30.976
C05023=1012.846,45.975,379.086,-28.812,53.703,-31.001
C05024=1012.850,45.579,379.116,-28.801,53.558,-31.026
C05025=1012.854,45.184,379.147,-28.790,53.413,-31.050
C05026=1012.859,44.788,379.178,-28.779,53.269,-31.075
C05027=1012.862,44.392,379.209,-28.769,53.125,-31.100
C05028=1012.866,43.997,379.239,-28.758,52.982,-31.126
C05029=1012.871,43.601,379.271,-28.747,52.838,-31.151
C05030=1012.875,43.205,379.301,-28.736,52.696,-31.178
C05031=1012.879,42.810,379.332,-28.726,52.553,-31.204
C05032=1012.883,42.415,379.363,-28.715,52.412,-31.230
C05033=1012.887,42.019,379.394,-28.704,52.270,-31.256
C05034=1012.891,41.624,379.425,-28.694,52.131,-31.282
C05035=1012.896,41.228,379.455,-28.683,51.990,-31.310
C05036=1012.899,40.833,379.486,-28.672,51.850,-31.336
C05037=1012.904,40.437,379.517,-28.662,51.711,-31.363
C05038=1012.908,40.042,379.548,-28.651,51.572,-31.390
C05039=1012.912,39.646,379.579,-28.641,51.435,-31.417
C05040=1012.916,39.250,379.609,-28.630,51.297,-31.445
C05041=1012.921,38.855,379.640,-28.620,51.159,-31.472
C05042=1012.924,38.460,379.671,-28.609,51.023,-31.500
C05043=1012.928,38.065,379.702,-28.599,50.888,-31.527
C05044=1012.932,37.669,379.732,-28.588,50.752,-31.556
C05045=1012.936,37.274,379.763,-28.578,50.617,-31.583
C05046=1012.941,36.878,379.795,-28.567,50.483,-31.612
C05047=1012.945,36.483,379.825,-28.557,50.349,-31.640
C05048=1012.949,36.088,379.856,-28.546,50.214,-31.669
C05049=1012.953,35.693,379.887,-28.536,50.081,-31.697
C05050=1012.956,35.297,379.918,-28.526,49.950,-31.726
C05051=1012.961,34.902,379.949,-28.515,49.817,-31.754
C05052=1012.965,34.506,379.979,-28.505,49.686,-31.784
C05053=1012.969,34.111,380.011,-28.494,49.555,-31.812
C05054=1012.973,33.716,380.041,-28.484,49.425,-31.841
C05055=1012.977,33.321,380.072,-28.474,49.294,-31.871
C05056=1012.981,32.926,380.103,-28.463,49.165,-31.899
C05057=1012.984,32.530,380.134,-28.453,49.036,-31.929
C05058=1012.988,32.135,380.165,-28.443,48.908,-31.959
C05059=1012.993,31.740,380.195,-28.432,48.780,-31.988
C05060=1012.997,31.344,380.227,-28.422,48.654,-32.018
C05061=1013.001,30.949,380.258,-28.412,48.526,-32.048
C05062=1013.005,30.554,380.289,-28.401,48.400,-32.077
C05063=1013.009,30.159,380.320,-28.391,48.274,-32.108
C05064=1013.012,29.763,380.351,-28.381,48.149,-32.138
C05065=1013.016,29.368,380.382,-28.370,48.025,-32.167
C05066=1013.020,28.973,380.412,-28.360,47.900,-32.198
C05067=1013.024,28.578,380.443,-28.350,47.777,-32.228
C05068=1013.027,28.184,380.474,-28.339,47.655,-32.258
C05069=1013.032,27.791,380.505,-28.329,47.533,-32.288
C05070=1013.036,27.398,380.536,-28.319,47.412,-32.318
C05071=1013.039,27.005,380.567,-28.309,47.292,-32.348
C05072=1013.043,26.611,380.598,-28.298,47.172,-32.379
C05073=1013.047,26.214,380.628,-28.288,47.051,-32.409
C05074=1013.051,25.817,380.660,-28.278,46.931,-32.440
C05075=1013.054,25.418,380.691,-28.268,46.811,-32.472
C05076=1013.057,25.023,380.722,-28.257,46.693,-32.502
C05077=1013.061,24.628,380.753,-28.247,46.574,-32.533
C05078=1013.066,24.231,380.784,-28.237,46.458,-32.563
C05079=1013.069,23.852,380.814,-28.227,46.346,-32.593
C05080=1013.072,23.512,380.840,-28.218,46.246,-32.620
C05081=1013.076,23.097,380.873,-28.208,46.126,-32.652
C05082=1013.079,22.733,380.902,-28.198,46.019,-32.680
C05083=1013.082,22.456,380.923,-28.191,45.939,-32.702
C05084=1013.085,22.124,380.949,-28.182,45.844,-32.728
C05085=1013.088,21.796,380.975,-28.174,45.750,-32.754
C05086=1013.092,21.408,381.005,-28.164,45.639,-32.783
C05087=1013.093,21.180,381.023,-28.158,45.575,-32.802
C05088=1013.096,20.932,381.043,-28.152,45.504,-32.822
C05089=1013.099,20.672,381.063,-28.145,45.430,-32.841
C05090=1013.101,20.404,381.084,-28.138,45.356,-32.862
C05091=1013.103,20.135,381.105,-28.131,45.280,-32.883
C05092=1013.105,19.874,381.125,-28.125,45.207,-32.903
C05093=1013.108,19.631,381.145,-28.119,45.140,-32.922
C05094=1013.110,19.411,381.161,-28.113,45.079,-32.940
C05095=1013.111,19.208,381.178,-28.108,45.023,-32.955
C05096=1013.116,18.806,381.210,-28.098,44.912,-32.987
C05097=1013.119,18.406,381.240,-28.087,44.803,-33.018
C05098=1013.122,18.014,381.272,-28.078,44.697,-33.049
C05099=1013.126,17.620,381.302,-28.067,44.589,-33.080
C05100=1013.129,17.236,381.333,-28.058,44.486,-33.110
C05101=1013.132,16.850,381.363,-28.048,44.383,-33.140
C05102=1013.136,16.466,381.393,-28.038,44.282,-33.169
C05103=1013.139,16.083,381.423,-28.029,44.180,-33.200
C05104=1013.142,15.703,381.453,-28.019,44.080,-33.229
C05105=1013.146,15.321,381.483,-28.009,43.981,-33.258
C05106=1013.149,14.942,381.513,-28.000,43.883,-33.288
C05107=1013.152,14.562,381.543,-27.990,43.785,-33.318
C05108=1013.155,14.182,381.572,-27.981,43.686,-33.348
C05109=1013.158,13.801,381.602,-27.971,43.589,-33.377
C05110=1013.162,13.419,381.632,-27.962,43.493,-33.407
C05111=1013.165,13.037,381.662,-27.952,43.397,-33.437
C05112=1013.167,12.653,381.692,-27.943,43.301,-33.465
C05113=1013.171,12.269,381.722,-27.933,43.205,-33.495
C05114=1013.175,11.887,381.752,-27.924,43.111,-33.524
C05115=1013.177,11.515,381.782,-27.915,43.020,-33.554
C05116=1013.181,11.152,381.810,-27.906,42.931,-33.582
C05117=1013.183,10.787,381.839,-27.897,42.842,-33.609
C05118=1013.186,10.413,381.868,-27.888,42.752,-33.638
C05119=1013.189,10.035,381.898,-27.878,42.662,-33.667
C05120=1013.193,9.659,381.928,-27.869,42.572,-33.696
C05121=1013.195,9.285,381.957,-27.860,42.483,-33.724
C05122=1013.198,8.911,381.987,-27.851,42.396,-33.753
C05123=1013.201,8.537,382.016,-27.842,42.309,-33.780
C05124=1013.204,8.164,382.045,-27.833,42.221,-33.809
C05125=1013.207,7.788,382.074,-27.824,42.136,-33.838
C05126=1013.210,7.409,382.104,-27.815,42.050,-33.866
C05127=1013.213,7.028,382.133,-27.806,41.963,-33.895
C05128=1013.216,6.643,382.164,-27.796,41.876,-33.922
C05129=1013.218,6.252,382.195,-27.787,41.789,-33.952
C05130=1013.222,5.859,382.226,-27.778,41.702,-33.981
C05131=1013.224,5.467,382.257,-27.769,41.615,-34.011
C05132=1013.228,5.076,382.288,-27.759,41.529,-34.040
C05133=1013.231,4.688,382.318,-27.750,41.445,-34.067
C05134=1013.233,4.298,382.349,-27.741,41.361,-34.096
C05135=1013.236,3.907,382.379,-27.732,41.278,-34.126
C05136=1013.239,3.535,382.409,-27.723,41.199,-34.152
C05137=1013.241,3.191,382.436,-27.715,41.125,-34.178
C05138=1013.243,2.868,382.461,-27.708,41.058,-34.200
C05139=1013.246,2.545,382.486,-27.701,40.991,-34.224
C05140=1013.248,2.203,382.514,-27.693,40.921,-34.249
C05141=1013.251,1.832,382.542,-27.684,40.845,-34.275
C05142=1013.253,1.439,382.573,-27.675,40.765,-34.304
C05143=1013.256,1.042,382.604,-27.666,40.685,-34.331
C05144=1013.259,0.646,382.635,-27.657,40.606,-34.361
C05145=1013.261,0.251,382.667,-27.649,40.528,-34.388
C05146=1013.264,-0.143,382.698,-27.640,40.450,-34.417
C05147=1013.267,-0.540,382.729,-27.631,40.372,-34.444
C05148=1013.270,-0.941,382.760,-27.622,40.296,-34.472
C05149=1013.272,-1.344,382.792,-27.613,40.219,-34.499
C05150=1013.274,-1.748,382.824,-27.605,40.142,-34.527
C05151=1013.277,-2.154,382.855,-27.596,40.066,-34.555
C05152=1013.280,-2.563,382.887,-27.587,39.990,-34.584
C05153=1013.283,-2.973,382.919,-27.578,39.914,-34.612
C05154=1013.285,-3.384,382.952,-27.569,39.839,-34.639
C05155=1013.287,-3.786,382.983,-27.561,39.766,-34.666
C05156=1013.290,-4.171,383.014,-27.553,39.698,-34.692
C05157=1013.293,-4.550,383.043,-27.545,39.631,-34.718
C05158=1013.295,-4.941,383.074,-27.537,39.562,-34.745
C05159=1013.297,-5.355,383.106,-27.528,39.490,-34.771
C05160=1013.299,-5.569,383.123,-27.524,39.453,-34.785
C05161=1013.299,-5.786,383.140,-27.519,39.417,-34.799
C05162=1013.301,-6.002,383.158,-27.515,39.379,-34.814
C05163=1013.302,-6.219,383.174,-27.510,39.343,-34.827
C05164=1013.304,-6.436,383.191,-27.506,39.307,-34.841
C05165=1013.304,-6.653,383.208,-27.502,39.270,-34.856
C05166=1013.306,-6.869,383.225,-27.497,39.233,-34.870
C05167=1013.307,-7.084,383.242,-27.493,39.198,-34.884
C05168=1013.308,-7.299,383.259,-27.489,39.163,-34.897
C05169=1013.309,-7.513,383.276,-27.484,39.127,-34.911
C05170=1013.311,-7.726,383.293,-27.480,39.093,-34.924
C05171=1013.312,-7.939,383.310,-27.476,39.058,-34.938
C05172=1013.313,-8.152,383.326,-27.472,39.024,-34.951
C05173=1013.314,-8.364,383.342,-27.468,38.991,-34.965
C05174=1013.316,-8.576,383.359,-27.464,38.957,-34.977
C05175=1013.317,-8.786,383.375,-27.460,38.924,-34.991
C05176=1013.318,-8.998,383.392,-27.456,38.891,-35.004
C05177=1013.320,-9.419,383.426,-27.447,38.825,-35.031
C05178=1013.322,-9.841,383.458,-27.440,38.761,-35.056
C05179=1013.325,-10.262,383.492,-27.432,38.697,-35.082
C05180=1013.327,-10.682,383.525,-27.424,38.633,-35.108
C05181=1013.329,-11.101,383.557,-27.416,38.571,-35.132
C05182=1013.331,-11.518,383.590,-27.408,38.511,-35.157
C05183=1013.333,-11.935,383.622,-27.401,38.451,-35.181
C05184=1013.335,-12.350,383.655,-27.393,38.391,-35.206
C05185=1013.337,-12.762,383.687,-27.386,38.334,-35.230
C05186=1013.339,-13.171,383.720,-27.379,38.277,-35.253
C05187=1013.341,-13.570,383.750,-27.372,38.223,-35.274
C05188=1013.343,-13.956,383.781,-27.365,38.171,-35.296
C05189=1013.345,-14.334,383.810,-27.359,38.120,-35.318
C05190=1013.347,-14.708,383.839,-27.353,38.071,-35.340
C05191=1013.349,-15.085,383.869,-27.346,38.022,-35.361
C05192=1013.350,-15.468,383.899,-27.340,37.974,-35.382
C05193=1013.352,-15.860,383.929,-27.334,37.924,-35.404
C05194=1013.353,-16.257,383.961,-27.327,37.875,-35.424
C05195=1013.355,-16.651,383.991,-27.321,37.827,-35.445
C05196=1013.357,-17.050,384.023,-27.315,37.779,-35.465
C05197=1013.359,-17.444,384.054,-27.309,37.732,-35.485
C05198=1013.360,-17.831,384.083,-27.303,37.686,-35.506
C05199=1013.361,-18.034,384.099,-27.300,37.663,-35.517
C05200=1013.362,-18.260,384.118,-27.296,37.637,-35.528
C05201=1013.362,-18.513,384.137,-27.292,37.609,-35.540
C05202=1013.365,-18.785,384.159,-27.288,37.579,-35.554
C05203=1013.366,-19.064,384.180,-27.284,37.547,-35.567
C05204=1013.366,-19.338,384.202,-27.280,37.517,-35.582
C05205=1013.367,-19.594,384.221,-27.277,37.490,-35.594
C05206=1013.368,-19.825,384.239,-27.273,37.464,-35.605
C05207=1013.369,-20.031,384.255,-27.270,37.443,-35.616
C05208=1013.371,-20.381,384.282,-27.266,37.406,-35.631
C05209=1013.372,-20.778,384.314,-27.260,37.365,-35.650
C05210=1013.373,-21.170,384.344,-27.255,37.326,-35.669
C05211=1013.374,-21.564,384.375,-27.250,37.287,-35.687
C05212=1013.376,-21.957,384.406,-27.244,37.248,-35.705
C05213=1013.378,-22.350,384.437,-27.239,37.210,-35.722
C05214=1013.379,-22.743,384.468,-27.234,37.174,-35.740
C05215=1013.379,-23.136,384.498,-27.229,37.138,-35.757
C05216=1013.382,-23.530,384.529,-27.225,37.103,-35.774
C05217=1013.383,-23.923,384.559,-27.220,37.068,-35.791
C05218=1013.383,-24.316,384.590,-27.215,37.033,-35.808
C05219=1013.384,-24.709,384.620,-27.211,37.000,-35.824
C05220=1013.386,-25.102,384.652,-27.206,36.968,-35.841
C05221=1013.387,-25.495,384.682,-27.202,36.937,-35.856
C05222=1013.388,-25.889,384.712,-27.198,36.905,-35.871
C05223=1013.389,-26.282,384.743,-27.194,36.875,-35.887
C05224=1013.391,-26.675,384.774,-27.190,36.846,-35.902
C05225=1013.392,-27.069,384.805,-27.186,36.817,-35.917
C05226=1013.393,-27.461,384.835,-27.182,36.789,-35.931
C05227=1013.393,-27.855,384.866,-27.178,36.761,-35.945
C05228=1013.395,-28.248,384.896,-27.174,36.735,-35.960
C05229=1013.395,-28.642,384.927,-27.171,36.709,-35.974
C05230=1013.397,-29.034,384.957,-27.167,36.684,-35.987
C05231=1013.397,-29.428,384.988,-27.164,36.661,-36.000
C05232=1013.398,-29.821,385.019,-27.161,36.637,-36.013
C05233=1013.399,-30.214,385.049,-27.157,36.614,-36.026
C05234=1013.400,-30.608,385.080,-27.154,36.592,-36.039
C05235=1013.400,-31.001,385.110,-27.151,36.571,-36.051
C05236=1013.401,-31.395,385.141,-27.148,36.550,-36.064
C05237=1013.402,-31.788,385.172,-27.146,36.530,-36.075
C05238=1013.403,-32.181,385.202,-27.143,36.512,-36.086
C05239=1013.404,-32.575,385.233,-27.140,36.493,-36.098
C05240=1013.404,-32.969,385.263,-27.138,36.476,-36.110
C05241=1013.405,-33.361,385.294,-27.136,36.459,-36.120
C05242=1013.406,-33.755,385.325,-27.133,36.443,-36.130
C05243=1013.406,-34.148,385.355,-27.131,36.428,-36.141
C05244=1013.406,-34.541,385.386,-27.129,36.413,-36.150
C05245=1013.407,-34.935,385.416,-27.127,36.399,-36.160
C05246=1013.408,-35.329,385.447,-27.125,36.387,-36.169
C05247=1013.408,-35.722,385.477,-27.123,36.375,-36.178
C05248=1013.409,-36.115,385.508,-27.122,36.363,-36.187
C05249=1013.409,-36.508,385.538,-27.120,36.353,-36.195
C05250=1013.409,-36.901,385.569,-27.119,36.343,-36.204
C05251=1013.410,-37.295,385.599,-27.118,36.334,-36.212
C05252=1013.410,-37.688,385.630,-27.116,36.326,-36.219
C05253=1013.411,-38.082,385.660,-27.115,36.318,-36.227
C05254=1013.411,-38.476,385.691,-27.114,36.312,-36.234
C05255=1013.411,-38.869,385.721,-27.113,36.305,-36.241
C05256=1013.412,-39.262,385.752,-27.113,36.300,-36.248
C05257=1013.412,-39.655,385.782,-27.112,36.297,-36.255
C05258=1013.412,-40.048,385.812,-27.112,36.293,-36.259
C05259=1013.412,-40.441,385.843,-27.111,36.290,-36.265
C05260=1013.412,-40.834,385.873,-27.111,36.288,-36.272
C05261=1013.412,-41.227,385.903,-27.111,36.287,-36.276
C05262=1013.413,-41.621,385.934,-27.111,36.286,-36.281
C05263=1013.412,-42.014,385.964,-27.111,36.286,-36.287
C05264=1013.412,-42.406,385.995,-27.111,36.287,-36.292
C05265=1013.412,-42.800,386.025,-27.111,36.289,-36.295
C05266=1013.412,-43.192,386.055,-27.111,36.292,-36.298
C05267=1013.412,-43.585,386.086,-27.112,36.295,-36.302
C05268=1013.413,-43.979,386.116,-27.113,36.300,-36.305
C05269=1013.413,-44.372,386.147,-27.113,36.304,-36.308
C05270=1013.412,-44.764,386.178,-27.114,36.310,-36.312
C05271=1013.412,-45.157,386.208,-27.115,36.316,-36.314
C05272=1013.412,-45.550,386.238,-27.116,36.324,-36.315
C05273=1013.411,-45.943,386.267,-27.117,36.332,-36.316
C05274=1013.411,-46.335,386.298,-27.118,36.341,-36.318
C05275=1013.411,-46.728,386.329,-27.120,36.351,-36.319
C05276=1013.411,-47.121,386.359,-27.121,36.362,-36.321
C05277=1013.411,-47.513,386.389,-27.123,36.372,-36.321
C05278=1013.410,-47.906,386.419,-27.125,36.385,-36.322
C05279=1013.410,-48.299,386.449,-27.127,36.398,-36.323
C05280=1013.409,-48.692,386.480,-27.129,36.411,-36.322
C05281=1013.409,-49.084,386.510,-27.131,36.426,-36.320
C05282=1013.409,-49.476,386.540,-27.133,36.442,-36.321
C05283=1013.408,-49.869,386.571,-27.135,36.458,-36.320
C05284=1013.407,-50.262,386.601,-27.138,36.474,-36.318
C05285=1013.408,-50.654,386.631,-27.140,36.492,-36.316
C05286=1013.406,-51.046,386.661,-27.143,36.511,-36.315
C05287=1013.406,-51.439,386.692,-27.146,36.530,-36.312
C05288=1013.405,-51.832,386.722,-27.148,36.550,-36.310
C05289=1013.405,-52.225,386.752,-27.151,36.571,-36.307
C05290=1013.404,-52.617,386.783,-27.155,36.593,-36.304
C05291=1013.403,-53.009,386.812,-27.158,36.615,-36.300
C05292=1013.403,-53.402,386.843,-27.161,36.639,-36.296
C05293=1013.402,-53.794,386.872,-27.165,36.662,-36.292
C05294=1013.401,-54.187,386.903,-27.168,36.687,-36.288
C05295=1013.400,-54.579,386.933,-27.172,36.713,-36.284
C05296=1013.400,-54.971,386.963,-27.176,36.740,-36.279
C05297=1013.399,-55.363,386.993,-27.180,36.767,-36.274
C05298=1013.398,-55.756,387.023,-27.184,36.795,-36.268
C05299=1013.397,-56.148,387.053,-27.188,36.825,-36.262
C05300=1013.397,-56.541,387.084,-27.192,36.854,-36.257
C05301=1013.395,-56.935,387.114,-27.197,36.885,-36.251
C05302=1013.394,-57.328,387.143,-27.201,36.916,-36.244
C05303=1013.393,-57.722,387.174,-27.206,36.949,-36.237
C05304=1013.392,-58.116,387.205,-27.210,36.982,-36.231
C05305=1013.392,-58.511,387.235,-27.215,37.016,-36.223
C05306=1013.391,-58.906,387.265,-27.220,37.051,-36.216
C05307=1013.389,-59.302,387.296,-27.225,37.087,-36.207
C05308=1013.387,-59.698,387.326,-27.231,37.124,-36.199
C05309=1013.387,-60.095,387.357,-27.236,37.162,-36.190
C05310=1013.385,-60.491,387.387,-27.241,37.200,-36.181
C05311=1013.384,-60.889,387.417,-27.247,37.239,-36.173
C05312=1013.383,-61.288,387.447,-27.253,37.280,-36.162
C05313=1013.381,-61.686,387.479,-27.259,37.321,-36.153
C05314=1013.380,-62.086,387.508,-27.264,37.363,-36.143
C05315=1013.379,-62.485,387.540,-27.271,37.406,-36.132
C05316=1013.378,-62.886,387.570,-27.277,37.450,-36.122
C05317=1013.376,-63.287,387.601,-27.283,37.495,-36.110
C05318=1013.375,-63.688,387.631,-27.289,37.541,-36.099
C05319=1013.373,-64.089,387.662,-27.296,37.587,-36.088
C05320=1013.371,-64.492,387.693,-27.303,37.635,-36.076
C05321=1013.370,-64.894,387.723,-27.310,37.684,-36.064
C05322=1013.369,-65.296,387.755,-27.316,37.733,-36.052
C05323=1013.367,-65.699,387.785,-27.323,37.783,-36.038
C05324=1013.366,-66.103,387.816,-27.331,37.834,-36.025
C05325=1013.363,-66.506,387.847,-27.338,37.886,-36.012
C05326=1013.363,-66.909,387.878,-27.345,37.939,-35.998
C05327=1013.360,-67.313,387.908,-27.353,37.994,-35.985
C05328=1013.359,-67.717,387.940,-27.360,38.049,-35.970
C05329=1013.357,-68.121,387.971,-27.368,38.104,-35.956
C05330=1013.355,-68.525,388.002,-27.376,38.160,-35.942
C05331=1013.353,-68.929,388.033,-27.384,38.217,-35.927
C05332=1013.352,-69.334,388.064,-27.392,38.277,-35.912
C05333=1013.350,-69.738,388.094,-27.400,38.336,-35.897
C05334=1013.348,-70.142,388.125,-27.408,38.396,-35.880
C05335=1013.346,-70.547,388.157,-27.416,38.457,-35.864
C05336=1013.344,-70.951,388.187,-27.425,38.518,-35.848
C05337=1013.342,-71.355,388.218,-27.433,38.581,-35.831
C05338=1013.340,-71.759,388.249,-27.442,38.644,-35.815
C05339=1013.339,-72.163,388.280,-27.451,38.709,-35.798
C05340=1013.336,-72.567,388.311,-27.460,38.775,-35.781
C05341=1013.334,-72.970,388.341,-27.469,38.841,-35.763
C05342=1013.332,-73.374,388.371,-27.478,38.908,-35.746
C05343=1013.330,-73.777,388.403,-27.487,38.976,-35.727
C05344=1013.328,-74.181,388.433,-27.496,39.046,-35.710
C05345=1013.326,-74.584,388.464,-27.506,39.115,-35.692
C05346=1013.324,-74.987,388.495,-27.515,39.186,-35.671
C05347=1013.321,-75.389,388.526,-27.525,39.258,-35.653
C05348=1013.319,-75.792,388.556,-27.534,39.330,-35.634
C05349=1013.317,-76.195,388.587,-27.544,39.403,-35.615
C05350=1013.315,-76.597,388.618,-27.554,39.477,-35.595
C05351=1013.313,-77.000,388.648,-27.564,39.552,-35.576
C05352=1013.311,-77.402,388.679,-27.574,39.628,-35.555
C05353=1013.308,-77.804,388.710,-27.584,39.704,-35.535
C05354=1013.305,-78.205,388.740,-27.594,39.782,-35.514
C05355=1013.303,-78.606,388.771,-27.604,39.860,-35.493
C05356=1013.301,-79.007,388.801,-27.615,39.939,-35.473
C05357=1013.299,-79.407,388.832,-27.625,40.019,-35.452
C05358=1013.295,-79.807,388.862,-27.635,40.099,-35.430
C05359=1013.293,-80.206,388.893,-27.646,40.181,-35.408
C05360=1013.291,-80.605,388.923,-27.657,40.264,-35.387
C05361=1013.288,-81.003,388.954,-27.667,40.346,-35.366
C05362=1013.285,-81.399,388.984,-27.678,40.429,-35.344
C05363=1013.284,-81.797,389.014,-27.689,40.514,-35.321
C05364=1013.281,-82.196,389.045,-27.700,40.599,-35.300
C05365=1013.278,-82.594,389.075,-27.711,40.686,-35.276
C05366=1013.276,-82.989,389.105,-27.722,40.773,-35.254
C05367=1013.273,-83.386,389.135,-27.733,40.860,-35.231
C05368=1013.271,-83.782,389.165,-27.745,40.949,-35.208
C05369=1013.268,-84.173,389.195,-27.756,41.037,-35.186
C05370=1013.265,-84.565,389.225,-27.767,41.127,-35.162
C05371=1013.262,-84.984,389.257,-27.779,41.223,-35.137
C05372=1013.260,-85.213,389.274,-27.786,41.276,-35.123
C05373=1013.259,-85.451,389.292,-27.793,41.331,-35.110
C05374=1013.257,-85.690,389.311,-27.800,41.387,-35.095
C05375=1013.256,-85.925,389.329,-27.807,41.443,-35.081
C05376=1013.254,-86.147,389.346,-27.813,41.496,-35.068
C05377=1013.251,-86.555,389.376,-27.825,41.592,-35.042
C05378=1013.248,-86.943,389.406,-27.837,41.687,-35.018
C05379=1013.246,-87.320,389.435,-27.848,41.778,-34.994
C05380=1013.243,-87.688,389.463,-27.859,41.868,-34.972
C05381=1013.241,-88.050,389.491,-27.870,41.958,-34.949
C05382=1013.238,-88.427,389.520,-27.882,42.051,-34.925
C05383=1013.235,-88.811,389.549,-27.894,42.148,-34.901
C05384=1013.234,-89.031,389.565,-27.900,42.203,-34.887
C05385=1013.232,-89.273,389.584,-27.908,42.264,-34.872
C05386=1013.230,-89.529,389.604,-27.916,42.330,-34.856
C05387=1013.228,-89.788,389.623,-27.924,42.397,-34.838
C05388=1013.226,-90.039,389.642,-27.932,42.461,-34.822
C05389=1013.224,-90.272,389.660,-27.939,42.522,-34.807
C05390=1013.222,-90.483,389.676,-27.946,42.577,-34.793
C05391=1013.220,-90.751,389.697,-27.954,42.648,-34.776
C05392=1013.217,-91.105,389.724,-27.966,42.741,-34.753
C05393=1013.214,-91.494,389.753,-27.978,42.845,-34.727
C05394=1013.211,-91.883,389.783,-27.991,42.949,-34.702
C05395=1013.208,-92.271,389.813,-28.003,43.053,-34.676
C05396=1013.205,-92.658,389.842,-28.016,43.159,-34.650
C05397=1013.202,-93.045,389.871,-28.028,43.265,-34.624
C05398=1013.199,-93.430,389.901,-28.041,43.372,-34.598
C05399=1013.196,-93.816,389.930,-28.053,43.478,-34.572
C05400=1013.193,-94.200,389.959,-28.066,43.586,-34.546
C05401=1013.189,-94.582,389.989,-28.079,43.696,-34.520
C05402=1013.187,-94.964,390.018,-28.091,43.803,-34.494
C05403=1013.184,-95.345,390.047,-28.104,43.913,-34.467
C05404=1013.180,-95.723,390.075,-28.117,44.023,-34.441
C05405=1013.178,-96.102,390.104,-28.130,44.132,-34.415
C05406=1013.174,-96.479,390.133,-28.142,44.243,-34.389
C05407=1013.171,-96.855,390.161,-28.155,44.354,-34.364
C05408=1013.168,-97.231,390.191,-28.168,44.466,-34.338
C05409=1013.165,-97.607,390.219,-28.181,44.578,-34.310
C05410=1013.161,-97.982,390.248,-28.194,44.691,-34.285
C05411=1013.158,-98.357,390.277,-28.207,44.806,-34.259
C05412=1013.156,-98.734,390.305,-28.220,44.921,-34.232
C05413=1013.152,-99.109,390.334,-28.233,45.035,-34.206
C05414=1013.149,-99.486,390.363,-28.246,45.153,-34.179
C05415=1013.146,-99.864,390.392,-28.260,45.271,-34.152
C05416=1013.142,-100.242,390.420,-28.273,45.388,-34.125
C05417=1013.138,-100.622,390.449,-28.286,45.509,-34.098
C05418=1013.135,-101.002,390.478,-28.300,45.629,-34.072
C05419=1013.133,-101.384,390.507,-28.313,45.751,-34.044
C05420=1013.129,-101.767,390.537,-28.327,45.874,-34.016
C05421=1013.126,-102.150,390.566,-28.341,45.999,-33.989
C05422=1013.122,-102.535,390.596,-28.355,46.124,-33.961
C05423=1013.118,-102.919,390.625,-28.369,46.251,-33.934
C05424=1013.115,-103.305,390.654,-28.383,46.378,-33.906
C05425=1013.112,-103.692,390.683,-28.397,46.507,-33.878
C05426=1013.108,-104.078,390.713,-28.411,46.635,-33.851
C05427=1013.105,-104.466,390.743,-28.425,46.766,-33.822
C05428=1013.101,-104.854,390.773,-28.440,46.897,-33.795
C05429=1013.098,-105.242,390.803,-28.454,47.029,-33.767
C05430=1013.094,-105.631,390.832,-28.468,47.163,-33.738
C05431=1013.090,-106.019,390.862,-28.483,47.297,-33.711
C05432=1013.087,-106.410,390.892,-28.497,47.432,-33.683
C05433=1013.083,-106.817,390.923,-28.513,47.575,-33.654
C05434=1013.081,-107.031,390.939,-28.521,47.649,-33.639
C05435=1013.079,-107.251,390.956,-28.529,47.726,-33.623
C05436=1013.076,-107.478,390.974,-28.537,47.807,-33.606
C05437=1013.075,-107.708,390.991,-28.546,47.888,-33.589
C05438=1013.073,-107.940,391.009,-28.555,47.970,-33.572
C05439=1013.070,-108.172,391.026,-28.563,48.052,-33.556
C05440=1013.068,-108.401,391.044,-28.572,48.135,-33.539
C05441=1013.066,-108.626,391.061,-28.581,48.216,-33.522
C05442=1013.064,-108.845,391.078,-28.589,48.294,-33.507
C05443=1013.060,-109.262,391.111,-28.605,48.444,-33.477
C05444=1013.056,-109.657,391.140,-28.620,48.587,-33.449
C05445=1013.053,-110.046,391.170,-28.635,48.728,-33.422
C05446=1013.049,-110.434,391.200,-28.650,48.871,-33.395
C05447=1013.045,-110.822,391.229,-28.665,49.014,-33.367
C05448=1013.042,-111.211,391.259,-28.680,49.158,-33.340
C05449=1013.038,-111.600,391.289,-28.695,49.303,-33.312
C05450=1013.034,-111.989,391.319,-28.711,49.448,-33.285
C05451=1013.031,-112.377,391.349,-28.726,49.594,-33.257
C05452=1013.027,-112.766,391.379,-28.741,49.741,-33.231
C05453=1013.023,-113.155,391.408,-28.756,49.889,-33.203
C05454=1013.020,-113.542,391.438,-28.772,50.037,-33.176
C05455=1013.016,-113.931,391.468,-28.787,50.186,-33.149
C05456=1013.011,-114.319,391.498,-28.803,50.335,-33.123
